// TwinCAT 3 PLC project SPS_3
// ProgramVersion: 3.1.4026.10
// CompilerDefines: VISU_USEPROPERTYINFO
// libraries:
//   Tc2_ModbusRTU, * (Beckhoff Automation GmbH)
//   Tc2_Standard, * (Beckhoff Automation GmbH)
//   Tc2_System, * (Beckhoff Automation GmbH)
//   Tc2_TcpIp, * (Beckhoff Automation GmbH)
//   Tc2_Utilities, * (Beckhoff Automation GmbH)
// project tree:
//   DUTs/01_Listen/01_Zustände/ eObjectAktorState.TcDUT, eObjectSensorState.TcDUT, eSkillState.TcDUT, eSystemState.TcDUT
//   DUTs/01_Listen/02_Commands/ eSystemCommand.TcDUT
//   DUTs/01_Listen/03_Konfigurationen/ eRobMoveType.TcDUT, eRobPosType.TcDUT
//   DUTs/02_Schnittstellen/01_Skills/ I_Skill.TcIO (not stored), I_Skill_RoboterErweitert.TcIO, I_Skill_SmartGreifer.TcIO, I_Skill_Roboter.TcIO
//   DUTs/02_Schnittstellen/02_Objekte/ I_Objekt_Kraftsensor.TcIO (not stored), I_Objekt_Roboter.TcIO, I_Objekt_SmartGreifer.TcIO
//   DUTs/02_Schnittstellen/03_Sequenz/ I_Sequenz.TcIO
//   DUTs/03_Strukturen/01_Prozessparameter/ sKraftVariablen.TcDUT, sRoboterProzessVariablen.TcDUT, sSmartGreiferProzessVariablen.TcDUT
//   DUTs/03_Strukturen/02_Objektintern/01_FB_Roboter/ sPositionArrays.TcDUT, sPositionValues.TcDUT, sRealTimeData.TcDUT
//   DUTs/03_Strukturen/02_Objektintern/02_FB_Kraftsensor/ Kraftvariablen.TcDUT, Request.TcDUT, Response_Parameters.TcDUT, Response_Values.TcDUT
//   DUTs/03_Strukturen/ SkillInfo.TcDUT
//   DUTs/04_Union/ Array2_Int.TcDUT, Array8_LReal.TcDUT, Int_2Byte.TcDUT, String_Array256.TcDUT
//   / GlobalTextList.TcGTLO, PlcTask.TcTTO, Visualization Manager.TcVMO (not stored), VISU_TASK.TcTTO
//   GVLs/ GVL.TcGVL
//   POUs/00_Funktionsbausteine/ FB_PulseTrigger.TcPOU
//   POUs/01_Prozessmodell/01_Skills/01_V1/00_Basis/ FB_Basis_Skill.TcPOU, FB_SkillReferenz.TcPOU
//   POUs/01_Prozessmodell/01_Skills/01_V1/01_Roboter/ Skill_Position_anfahren.TcPOU, Skill_Position_anfahren_erweitert.TcPOU (not stored)
//   POUs/01_Prozessmodell/01_Skills/01_V1/02_Greifer/ Skill_Greifer_Pos_Anfahren.TcPOU (not stored)
//   POUs/01_Prozessmodell/01_Skills/02_V2/01_Roboter/ FB_SkillBasis.TcPOU, Skill_R_P2P.TcPOU
//   POUs/01_Prozessmodell/02_Sequenzen/00_Basis/ FB_Basis.TcPOU
//   POUs/01_Prozessmodell/02_Sequenzen/01_Version_1/ Seq_Ausrichten.TcPOU, Seq_Ausrichten_MPlate.TcPOU, Seq_Ausrichten_Plates.TcPOU, Seq_Get_Part.TcPOU, Seq_Set_MPlate.TcPOU, Seq_Set_Plate_1.TcPOU (not stored), Seq_Set_Plate_2.TcPOU (not stored)
//   POUs/01_Prozessmodell/02_Sequenzen/02_Version_2/ Seq_Teile_Hohlen.TcPOU
//   POUs/01_Prozessmodell/03_Arbeitsplan/ AP_V1.TcPOU, AP_V2.TcPOU, AP_V2_1.TcPOU
//   POUs/01_Prozessmodell/ SkillSet.TcPOU
//   POUs/02_Anlagenmodell/01_Objektklassen/00_Referenz/ Basis_Objekt.TcPOU, FB_Basis_Objekt_Aktor.TcPOU, FB_Basis_Objekt_Sensor.TcPOU
//   POUs/02_Anlagenmodell/01_Objektklassen/ FB_Kraftsensor_V2.TcPOU, FB_Roboter.TcPOU, FB_SmartGreifer.TcPOU
//   POUs/02_Anlagenmodell/ Anlage.TcPOU
//   POUs/03_Systemmodell/ Systemparameter.TcPOU, Zustandshandling.TcPOU
//   POUs/ MAIN.TcPOU, PunkteZuweisung_Temp.TcPOU
//   VISUs/ Visualization.TcVIS
// real-time tasks:
//   TASK VISU_TASK: cycle T#200000us, priority 30, ADS port 351
//   TASK PlcTask2: cycle T#10ms, priority 22, ADS port 353
// I/O:
//   DEVICE Gerät 1 (EtherCAT), AmsNetId 147.87.172.51.2.1
//     Box 1 (BK1120)
// variable links:
//   SPS_3/SPS_3 Instance <-> Device 1 (EtherCAT)/Box 1 (BK1120)
//     PlcTask Inputs/Anlage.Gripper.Communication.InData/D[{0..21}] <-> Term 2 (KL6041)/Channel 1/Data In {0..21}  (22 links)
//     PlcTask Inputs/Anlage.Gripper.Communication.InData/Status <-> Term 2 (KL6041)/Channel 1/Status
//     PlcTask Outputs/Anlage.Gripper.Communication.OutData/Ctrl <-> Term 2 (KL6041)/Channel 1/Ctrl
//     PlcTask Outputs/Anlage.Gripper.Communication.OutData/D[{0..21}] <-> Term 2 (KL6041)/Channel 1/Data Out {0..21}  (22 links)

CONFIGURATION SPS_3
    RESOURCE PLC ON TwinCAT3
        TASK PlcTask(INTERVAL := T#10ms, PRIORITY := 22);
        TASK VISU_TASK(INTERVAL := T#200000us, PRIORITY := 30);
        PROGRAM MAIN WITH PlcTask : MAIN;
        PROGRAM VisuElems_Visu_Prg WITH VISU_TASK : VisuElems.Visu_Prg;
    END_RESOURCE
END_CONFIGURATION

// ---- DUTs/01_Listen/01_Zustände/eObjectAktorState.TcDUT
{attribute 'qualified_only'}
{attribute 'strict'}
{attribute 'to_string'}
TYPE eObjectAktorState :
(
	AUS 					:= 0,				// Das Objekt ist ausgeschalten
	BEREIT 					:= 1,				// Das Objekt ist eingeschalten und bereit
	MANUELL					:= 2,				// Das Objekt befindet sich im Manuell-Modus
	LAUFEND 				:= 3,				// Das Objekt ist aktiv
	ABGESCHLOSSEN_INTERN 	:= 4,				// Das Objekt hat den Prozess durchgeführt und hat selbständig gestoppt
	ABGESCHLOSSEN_EXTERN	:= 5,				// Das Objekt wurde durch den Skill gestoppt (ERREICHT / LIMIT)
	GESTOPPT 				:= 6,				// Das Objekt wurde durch das System gestoppt
	FEHLER					:= 7				// Es gibt einen Fehler bezüglich des Objektes
);
END_TYPE

// ---- DUTs/01_Listen/01_Zustände/eObjectSensorState.TcDUT
{attribute 'qualified_only'}
{attribute 'strict'}
{attribute 'to_string'}
TYPE eObjectSensorState :
(
	AUS 					:= 0,				// Das Objekt ist ausgeschalten
	LAUFEND 				:= 1,				// Das Objekt ist aktiv
	FEHLER					:= 2				// Es gibt einen Fehler bezüglich des Objektes
);
END_TYPE

// ---- DUTs/01_Listen/01_Zustände/eSkillState.TcDUT
{attribute 'qualified_only'}
{attribute 'strict'}
{attribute 'to_string'}
TYPE eSkillState :
(
	BEREIT	 		:= 0,				// Der Skill ist bereit einen Prozess auszuführen (Startzustand)
	LAUFEND 		:= 1,				// Der Skill führt einen Prozess aus
	ABGESCHLOSSEN 	:= 2,				// Der Prozess wurde abgeschlossen (Durch Objekt abgeschlossen)
	FEHLER			:= 3,				// Es gibt einen Fehler bezüglich des Prozesses 
	LIMITE			:= 4,				// Grenzwert wurde überschritten und Prozess wurde abgebrochen
	ERREICHT		:= 5				// Prozessziel wurde erreicht und Prozess wurde durch Skill beendet  
);	
END_TYPE

// ---- DUTs/01_Listen/01_Zustände/eSystemState.TcDUT
{attribute 'qualified_only'}
{attribute 'strict'}
{attribute 'to_string'}
TYPE eSystemState :
(
	AUS 			:= 0,				// Das System ist ausgeschalten
	BEREIT 			:= 1,				// Das System ist eingeschalten und bereit einen Prozess durchzuführen
	LAUFEND 		:= 2,				// Ein Prozess wird ausgeführt
	GESTOPPT		:= 3,				// Ein Prozess wurde gestoppt
	FEHLER			:= 4				// Es gibt einen Fehler im System 
);
END_TYPE

// ---- DUTs/01_Listen/02_Commands/eSystemCommand.TcDUT
{attribute 'qualified_only'}
{attribute 'strict'}
{attribute 'to_string'}
TYPE eSystemCommand :
(
	KEINE		:= 0,
	AUSCHALTEN 	:= 1,
	EINSCHALTEN := 2,
	STOPPEN		:= 3,
	RESETTEN	:= 4
);
END_TYPE

// ---- DUTs/01_Listen/03_Konfigurationen/eRobMoveType.TcDUT
{attribute 'qualified_only'}
{attribute 'strict'}
{attribute 'to_string'}
TYPE eRobMoveType :
(
	LinearToolSpace 			:= 0,		// Move to position (linear in tool-space)
	LinearJointSpace 			:= 1,		// Move to position (linear in joint-space)
	CircularToolSpace 			:= 2,		// Move Circular: Move to position (circular in tool-space)
	BlendCircularMoveLinear		:= 3		// Move Process
);
END_TYPE

// ---- DUTs/01_Listen/03_Konfigurationen/eRobPosType.TcDUT
{attribute 'qualified_only'}
{attribute 'strict'}
{attribute 'to_string'}
TYPE eRobPosType :
(
	Absolut := 0,			// Absolute Bewegung bezogen auf Basis-Koordinatensystem
	Relativ := 1			// Relative Bewegung bezogen auf aktuelle Position
);
END_TYPE

// ---- DUTs/03_Strukturen/01_Prozessparameter/sKraftVariablen.TcDUT
TYPE sKraftVariablen :
STRUCT
	Fx					:LREAL;							// Kraft in X-Richtung 
	Fy					:LREAL;							// Kraft in Y-Richtung 
	Fz					:LREAL;							// Kraft in Z-Richtung 
END_STRUCT
END_TYPE

// ---- DUTs/03_Strukturen/01_Prozessparameter/sRoboterProzessVariablen.TcDUT

TYPE sRoboterProzessVariablen :
STRUCT
	q1					:LREAL;				// X-Koordinate oder Gelenkwinkel 1
	q2					:LREAL;				// Y-Koordinate oder Gelenkwinkel 2
	q3					:LREAL;				// Z-Koordinate oder Gelenkwinkel 3
	q4					:LREAL;				// Orintierung um X-Achse oder Gelenkwinkel 4
	q5					:LREAL;				// Orientierung um Y-Achse oder Gelenkwinkel 5
	q6					:LREAL;				// Orientierung um Z-Achse oder Gelenkwinkel 6
	v					:LREAL;				// Geschwindigkeit
	a					:LREAL;				// Beschleunigung
	PosTyp				:eRobPosType;		// Position-Typ definieren (Absolut / Relativ)		
	MoveTyp				:eRobMoveType;		// Bewegungsart definieren (Linear / Circular etc.)
END_STRUCT
END_TYPE

// ---- DUTs/03_Strukturen/01_Prozessparameter/sSmartGreiferProzessVariablen.TcDUT
TYPE sSmartGreiferProzessVariablen :
STRUCT
	Pos				:USINT;			// Position von Greifer in mm
	Geschw			:USINT;			// Geschwindigkeit in %
	F				:USINT;			// Kraft in %
END_STRUCT
	
END_TYPE

// ---- DUTs/03_Strukturen/02_Objektintern/01_FB_Roboter/sPositionArrays.TcDUT
TYPE sPositionArrays :
STRUCT
	q1		: ARRAY[0..7] OF BYTE;
	q2		: ARRAY[0..7] OF BYTE;
	q3		: ARRAY[0..7] OF BYTE;
	q4		: ARRAY[0..7] OF BYTE;
	q5		: ARRAY[0..7] OF BYTE;
	q6		: ARRAY[0..7] OF BYTE;
END_STRUCT
END_TYPE

// ---- DUTs/03_Strukturen/02_Objektintern/01_FB_Roboter/sPositionValues.TcDUT
TYPE sPositionValues :
STRUCT
	q1			:LREAL;
	q2			:LREAL;
	q3			:LREAL;
	q4			:LREAL;
	q5			:LREAL;
	q6			:LREAL;
END_STRUCT
END_TYPE

// ---- DUTs/03_Strukturen/02_Objektintern/01_FB_Roboter/sRealTimeData.TcDUT
TYPE sRealTimeData :
STRUCT
	messageSize 				: ARRAY[0..3] OF BYTE;
	
	timestamp 					: ARRAY[0..7] OF BYTE;
	
	//qTarget 					: ARRAY[0..47] OF BYTE;
	qTargetQ1 					: ARRAY[0..7] OF BYTE;
	qTargetQ2 					: ARRAY[0..7] OF BYTE;
	qTargetQ3 					: ARRAY[0..7] OF BYTE;
	qTargetQ4 					: ARRAY[0..7] OF BYTE;
	qTargetQ5 					: ARRAY[0..7] OF BYTE;
	qTargetQ6 					: ARRAY[0..7] OF BYTE;
	
	qdTarget 					: ARRAY[0..47] OF BYTE;
	
	qddTarget 					: ARRAY[0..47] OF BYTE;
	
	iTarget 					: ARRAY[0..47] OF BYTE;
	
	mTarget 					: ARRAY[0..47] OF BYTE;
	
	//qActual 					: ARRAY[0..47] OF BYTE;
	qActualQ1 					: ARRAY[0..7] OF BYTE;
	qActualQ2 					: ARRAY[0..7] OF BYTE;
	qActualQ3 					: ARRAY[0..7] OF BYTE;
	qActualQ4 					: ARRAY[0..7] OF BYTE;
	qActualQ5 					: ARRAY[0..7] OF BYTE;
	qActualQ6 					: ARRAY[0..7] OF BYTE;
	
	//qdActual 					: ARRAY[0..47] OF BYTE;
	qdActualQ1 					: ARRAY[0..7] OF BYTE;
	qdActualQ2 					: ARRAY[0..7] OF BYTE;
	qdActualQ3 					: ARRAY[0..7] OF BYTE;
	qdActualQ4 					: ARRAY[0..7] OF BYTE;
	qdActualQ5 					: ARRAY[0..7] OF BYTE;
	qdActualQ6 					: ARRAY[0..7] OF BYTE;
	
	iActual 					: ARRAY[0..47] OF BYTE;
	
	toolAccelerometerValues 	: ARRAY[0..23] OF BYTE;
	
	unused_1					: ARRAY[0..119] OF BYTE;
	
	tcpForce 					: ARRAY[0..47] OF BYTE;
	
	//toolVector 					: ARRAY[0..47] OF BYTE;
	toolVectorQ1 				: ARRAY[0..7] OF BYTE;
	toolVectorQ2 				: ARRAY[0..7] OF BYTE;
	toolVectorQ3 				: ARRAY[0..7] OF BYTE;
	toolVectorQ4 				: ARRAY[0..7] OF BYTE;
	toolVectorQ5 				: ARRAY[0..7] OF BYTE;
	toolVectorQ6 				: ARRAY[0..7] OF BYTE;
	
	tcpSpeed 					: ARRAY[0..47] OF BYTE;
	
	digitalInputBits 			: ARRAY[0..7] OF BYTE;
	
	unused_2					: ARRAY[0..119] OF BYTE;
END_STRUCT
END_TYPE

// ---- DUTs/03_Strukturen/02_Objektintern/02_FB_Kraftsensor/Kraftvariablen.TcDUT

TYPE Kraftvariablen :
STRUCT
	Fx					:LREAL;							// Kraft in X-Richtung 
	Fy					:LREAL;							// Kraft in Y-Richtung 
	Fz					:LREAL;							// Kraft in Z-Richtung 
	Tx					:LREAL;							// Moment auf X-Achse 
	Ty					:LREAL;							// Moment auf Y-Achse 
	Tz					:LREAL;							// Moment auf Z-Achse 
END_STRUCT
END_TYPE

// ---- DUTs/03_Strukturen/02_Objektintern/02_FB_Kraftsensor/Request.TcDUT
TYPE Request :
STRUCT
	Command			:UINT;		// Value according to the command table
	Data			:ARRAY[0..18] OF UINT := [0];		
END_STRUCT
END_TYPE

// ---- DUTs/03_Strukturen/02_Objektintern/02_FB_Kraftsensor/Response_Parameters.TcDUT
TYPE Response_Parameters :
STRUCT
	Header				:UINT;			// Fixed 0x1234
	Unit_Force			:USINT;			// The unit of the calculated Force values
	Unit_Torque			:USINT;			// The unit of the calculated Torque values
	CPF					:UDINT;			// Counts per Force value
	CPT					:UDINT;			// Counts per Torque value
	ScaleFactorFx		:UINT;			// Additional scaling factor (for the Fx,Fy,Fz,Tx,Ty,Tz)
	ScaleFactorFy		:UINT;			// Additional scaling factor (for the Fx,Fy,Fz,Tx,Ty,Tz)
	ScaleFactorFz		:UINT;			// Additional scaling factor (for the Fx,Fy,Fz,Tx,Ty,Tz)
	ScaleFactorTx		:UINT;			// Additional scaling factor (for the Fx,Fy,Fz,Tx,Ty,Tz)
	ScaleFactorTy		:UINT;			// Additional scaling factor (for the Fx,Fy,Fz,Tx,Ty,Tz)
	ScaleFactorTz		:UINT;			// Additional scaling factor (for the Fx,Fy,Fz,Tx,Ty,Tz)
END_STRUCT
END_TYPE

// ---- DUTs/03_Strukturen/02_Objektintern/02_FB_Kraftsensor/Response_Values.TcDUT
TYPE Response_Values :
STRUCT
	Header				:UINT;			// Fixed 0x1234
	Status				:UINT;			// Status word of the sensor and Compute Box
	Fx					:INT;			// X-axis force in 32 bit Counts*
	Fy					:INT;			// Y-axis force in 32 bit Counts*
	Fz					:INT;			// Z-axis force in 32 bit Counts*
	Tx					:INT;			// X-axis torque in 32 bit Counts* (0 if not available)
	Ty					:INT;			// Y-axis torque in 32 bit Counts* (0 if not available)
	Tz					:INT;			// Z-axis torque in 32 bit Counts* (0 if not available)
END_STRUCT
END_TYPE

// ---- DUTs/03_Strukturen/SkillInfo.TcDUT
TYPE SkillInfo :
STRUCT
	iState			:eSkillState;
	Data			:sRoboterProzessVariablen;
	iStateObj		:eObjectAktorState;
	DataObj			:sRoboterProzessVariablen;
END_STRUCT
END_TYPE

// ---- DUTs/04_Union/Array2_Int.TcDUT
TYPE Array2_Int :
UNION
	arrByte 		:ARRAY[0..1] OF BYTE;
	sValue			:INT; 
END_UNION
END_TYPE

// ---- DUTs/04_Union/Array8_LReal.TcDUT
TYPE Array8_LReal :
UNION
	arrByte			:ARRAY[0..7] OF BYTE;
	rValue			:LREAL;
END_UNION
END_TYPE

// ---- DUTs/04_Union/Int_2Byte.TcDUT
TYPE Int_2Byte :
UNION
	sValue			:INT; 
	arrByte 		:ARRAY[0..1] OF BYTE;
END_UNION
END_TYPE

// ---- DUTs/04_Union/String_Array256.TcDUT
TYPE String_Array256 :
UNION
	sValue			:STRING; 
	arrByte 		:ARRAY[0..255] OF BYTE;
END_UNION
END_TYPE

// ---- GVLs/GVL.TcGVL
{attribute 'qualified_only'}
VAR_GLOBAL
	// Schnittstellenvariablen 
		// System: 
		SystemState								:eSystemState; 
		SystemCommand							:eSystemCommand; 
		ErrorID									:INT;
		
		// Kontrollvariablen: 
		Reset									:BOOL;
		Execute									:BOOL;
		
		// Prozessvariablen
		eKraftLimitValue						:sKraftVariablen;
		eKraftErreichtValue						:sKraftVariablen;
		
		
		// SkillStates
		
		// ObjectStates
		Robot_State								:eObjectAktorState;
		Greifer_State							:eObjectAktorState;
		Sensor_State							:eObjectSensorState;
		
		// Testvariablen
		CountSkillStart							:INT;
		CountSkill								:INT;
		CountObjectStart						:INT;
		CountObject								:INT;
		TestCount								:INT;
		MethodeState							:INT;
		SkillArray								:ARRAY[0..10] OF sRoboterProzessVariablen;
		ObjectArray								:ARRAY[0..10] OF STRING;
		skillInfo 								:ARRAY[0..50] OF SkillInfo;
		InfoCountSkill							:INT;
		PulseNrArray							:Array[0..10] OF INT;
END_VAR

// ---- DUTs/02_Schnittstellen/01_Skills/I_Skill_RoboterErweitert.TcIO
INTERFACE I_Skill_RoboterErweitert

METHOD M_Reset : BOOL
VAR_INPUT
END_VAR
END_METHOD

METHOD M_Start : BOOL
VAR_INPUT
END_VAR
END_METHOD

METHOD M_Stop : BOOL
VAR_INPUT
END_VAR
END_METHOD

PROPERTY P_Erreicht : sKraftVariablen
SET
END_SET
END_PROPERTY

PROPERTY P_Limit : sKraftVariablen
SET
END_SET
END_PROPERTY

PROPERTY P_RobotParam : sRoboterProzessVariablen
SET
END_SET
END_PROPERTY

PROPERTY P_State : eSkillState
GET
END_GET
END_PROPERTY

END_INTERFACE

// ---- DUTs/02_Schnittstellen/01_Skills/I_Skill_SmartGreifer.TcIO
INTERFACE I_Skill_SmartGreifer

METHOD M_Reset : BOOL
VAR_INPUT
END_VAR
END_METHOD

METHOD M_Start : BOOL
VAR_INPUT
END_VAR
END_METHOD

METHOD M_Stop : BOOL
VAR_INPUT
END_VAR
END_METHOD

PROPERTY P_SGripperParam : sSmartGreiferProzessVariablen
SET
END_SET
END_PROPERTY

PROPERTY P_State : eSkillState
GET
END_GET
END_PROPERTY

END_INTERFACE

// ---- DUTs/02_Schnittstellen/01_Skills/I_Skill_Roboter.TcIO
INTERFACE I_Skill_Roboter

METHOD M_Reset : BOOL
VAR_INPUT
END_VAR
END_METHOD

METHOD M_Start : BOOL
VAR_INPUT
END_VAR
END_METHOD

METHOD M_Stop : BOOL
VAR_INPUT
END_VAR
END_METHOD

PROPERTY P_RobotParam : sRoboterProzessVariablen
SET
END_SET
END_PROPERTY

PROPERTY P_State : eSkillState
GET
END_GET
END_PROPERTY

END_INTERFACE

// ---- DUTs/02_Schnittstellen/02_Objekte/I_Objekt_Roboter.TcIO
INTERFACE I_Objekt_Roboter

METHOD M_Reset : BOOL
VAR_INPUT
END_VAR
END_METHOD

METHOD M_Start : BOOL
VAR_INPUT
END_VAR
END_METHOD

METHOD M_Stop : BOOL
VAR_INPUT
END_VAR
END_METHOD

PROPERTY P_Prozessparameter : sRoboterProzessVariablen
SET
END_SET
END_PROPERTY

PROPERTY P_State : eObjectAktorState
GET
END_GET
END_PROPERTY

PROPERTY Test_Param : sRoboterProzessVariablen
GET
END_GET
END_PROPERTY

END_INTERFACE

// ---- DUTs/02_Schnittstellen/02_Objekte/I_Objekt_SmartGreifer.TcIO
INTERFACE I_Objekt_SmartGreifer

METHOD M_Reset : BOOL
VAR_INPUT
END_VAR
END_METHOD

METHOD M_Start : BOOL
VAR_INPUT
END_VAR
END_METHOD

METHOD M_Stop : BOOL
VAR_INPUT
END_VAR
END_METHOD

PROPERTY P_Prozessparameter : sSmartGreiferProzessVariablen
SET
END_SET
END_PROPERTY

PROPERTY P_State : eObjectAktorState
GET
END_GET
END_PROPERTY

END_INTERFACE

// ---- DUTs/02_Schnittstellen/03_Sequenz/I_Sequenz.TcIO
INTERFACE I_Sequenz

METHOD M_Reset : BOOL
VAR_INPUT
END_VAR
END_METHOD

METHOD M_Start : BOOL
VAR_INPUT
END_VAR
END_METHOD

METHOD M_Stop : BOOL
VAR_INPUT
END_VAR
END_METHOD

PROPERTY P_Finished : BOOL
GET
END_GET
END_PROPERTY

PROPERTY P_State : INT
GET
END_GET
END_PROPERTY

END_INTERFACE

// ---- POUs/MAIN.TcPOU
PROGRAM MAIN
VAR
END_VAR

// Aufrufen der Objekte
Anlage();
// Aufrufen der Skills (Im Moment nur für V1 verwendet)
//SkillSet();
// Aufrufen der Systenparameterzuweisung 
Systemparameter();
// Aufrunfen des Zustandshandlings
Zustandshandling();
// Temporäre Punktedatenbank
PunkteZuweisung_Temp();

// Aufrufen von Testablauf
AP_V2();

END_PROGRAM

// ---- POUs/02_Anlagenmodell/Anlage.TcPOU
PROGRAM Anlage
VAR_INPUT
	UR5				:FB_Roboter;
	Gripper			:FB_SmartGreifer;
	HEX_E_V2		:FB_Kraftsensor_V2;
END_VAR

VAR
END_VAR

UR5(
    eSysState := GVL.SystemState,
    eSysCommand := GVL.SystemCommand,
    sIP := '192.168.1.100',
    iPort_Prim := 30002,
    iPort_RT := 30003); // FB_Roboter
Gripper(eSysState := GVL.SystemState, eSysCommand := GVL.SystemCommand); // FB_SmartGreifer
HEX_E_V2(
    eSysState := GVL.SystemState,
    eSysCommand := GVL.SystemCommand,
    sIP := '192.168.1.10',
    iPort := 49151); // FB_Kraftsensor_V2

END_PROGRAM

// ---- POUs/02_Anlagenmodell/01_Objektklassen/FB_Roboter.TcPOU
FUNCTION_BLOCK FB_Roboter EXTENDS FB_Basis_Objekt_Aktor IMPLEMENTS I_Objekt_Roboter
VAR_INPUT
	// Kommunikationsvariablen
	sIP						:T_IPv4Addr;
	iPort_Prim				:UINT;
	iPort_RT				:UINT;
END_VAR

VAR_OUTPUT
END_VAR

VAR
	// Instanziierung von Kommunikationsbausteine
	Connect					:FB_SocketConnect;
	Disconnect				:FB_SocketCloseALL;
	Send_START				:FB_SocketSend;
	Send_STOP				:FB_SocketSend;
	Connect_RT				:FB_SocketConnect;
	Receive_RT				:FB_SocketReceive;
	Disconnect_RT			:FB_SocketClose;
	
	// Kommunikationsvariablen
	sSrvNetId   			:T_AmsNetId := '';
	tTimeout    			:TIME := T#45S;(*!!!*)
	hSocket    				:T_HSOCKET;
	hSocket_RT    			:T_HSOCKET;
	
	// Managementvariablen
	bEingeschalten 			:BOOL;
	bAusgeschalten			:BOOL;
	bAmStarten				:BOOL;
	bGestartet				:BOOL;
	bAmStoppen				:BOOL;
	bGestoppt				:BOOL;
	
	bStopCommand			:BOOL;
	bTurnedOn 				:BOOL;
	
	bBewegungStoppen		:BOOL;
	
	Delay_1					:TON;
	Execute_TON1			:BOOL;
	Delay_2					:TON;
	
	bQ1						:BOOL;
	bQ2						:BOOL;
	bQ3						:BOOL;
	bQ4						:BOOL;
	bQ5						:BOOL;
	bQ6						:BOOL;
	
	bVQ1					:BOOL;
	bVQ2					:BOOL;
	bVQ3					:BOOL;
	bVQ4					:BOOL;
	bVQ5					:BOOL;
	bVQ6					:BOOL;
	
	// RealTimeDatenerfassung
	RT_State				:INT;							// RealTime-State-Variable
	ReceivedData			:sRealTimedata;					// Erhaltene Daten von Roboter
	nRecBytes				:UDINT;							// Anzahl der erhaltenen Bytes
	
	JointPositions			:sPositionValues;				// Ausgelesene aktuelle Joint-Positonen-Byte
	JointSpeed				:sPositionValues;				// Ausgelesene aktuelle Joint-Geschwindigkeit-Byte
	ToolPosition			:sPositionValues;				// Ausgelesene aktuelle Tool-Positonen-Byte
	
	TempJointPosRev			:sPositionArrays;				// Ausgelesene aktuelle Joint-Positonen-Byte (Reversed)
	TempJointVRev			:sPositionArrays;				// Ausgelesene aktuelle Joint-Geschwindigkeit-Byte (Reversed)	
	TempToolPosRev			:sPositionArrays;				// Ausgelesene aktuelle Tool-Positonen-Byte(Reversed)
	
	Joint					:Array8_LReal;					// Aktuelle Joint-Positonen
	JSpeed					:Array8_LReal;					// Aktuelle Joint-Geschwindgeit
	Tool					:Array8_LReal;					// Aktuelle Tool-Positionen
	m						:INT;							// Loop-Variable
	
	// Prozessdaten
	TargetPosition			:sPositionValues;				// Targetpositions
	bSetValues				:BOOL;							// Definiert ob Targetposition noch ermittelt werden muss
	Prozessvariablen		:sRoboterProzessVariablen;
	
	Stateset				:BOOL;
END_VAR

// Instanziierungen
	Connect_RT(sSrvNetId := sSrvNetId,
							sRemoteHost := sIP,
							nRemotePort := iPort_RT,
							tTimeout := tTimeout,
							bError => bFehler,
							nErrId => iErrorID,
							hSocket => hSocket_RT);	
							
	Send_START(sSrvNetId := sSrvNetId,
			hSocket := hSocket,
			tTimeout := tTimeout,
			bError => bFehler,
			nErrId => iErrorID);
	Send_STOP(sSrvNetId := sSrvNetId,
			hSocket := hSocket,
			tTimeout := tTimeout,
			bError => bFehler,
			nErrId => iErrorID);
							
	Receive_RT(sSrvNetId := sSrvNetId,
							hSocket := hSocket_RT,
							cbLen := SIZEOF(ReceivedData),
							pDest := ADR(ReceivedData),
							tTimeout := tTimeout,
							bError => bFehler,
							nErrId => iErrorID,
							nRecBytes => nRecBytes);
							
	Disconnect_RT(sSrvNetId := sSrvNetId,
							hSocket := hSocket_RT,
							tTimeout := tTimeout,
							bError => bFehler,
							nErrId => iErrorID);
	
	Delay_1(IN := Execute_TON1, PT := T#3MS);
//____________________________________________________________________________________________
// Input-Command-Verwaltung
	// System
	IF eSysCommand = 2 AND iState = 0 THEN			// Objekt einschalten
		bEinschalten := TRUE;
	ELSE 
		bEinschalten := FALSE;
	END_IF
	
	IF eSysCommand = 1 AND iState = 1 THEN			// Objekt ausschalten
		bAusschalten := TRUE;		
	ELSE 
		bAusschalten := FALSE;		
	END_IF
	
	IF eSysCommand = 3 THEN							// Objekt beendet Prozess
		bStoppen := TRUE;
	ELSE
		bStoppen := FALSE;
	END_IF
	
	IF eSysCommand = 4 THEN							// System resettet Objekt
		bResettenSystem := TRUE;
	ELSE
		bResettenSystem := FALSE;
	END_IF
	
	
//____________________________________________________________________________________________
// Interner Methodenaufruf (Durch System oder Skill)
IF bEinschalten THEN
	bEingeschalten := M_Verbinden();
	bTurnedOn := TRUE;
ELSE 
	bEingeschalten := FALSE;
END_IF

IF bAusschalten THEN
	bAusgeschalten := M_Trennen();
	bTurnedOn := FALSE;
	RT_State := 0;
ELSE 
	bAusgeschalten := FALSE;
END_IF

//____________________________________________________________________________________________
// Datenerfassungsprozess
IF bTurnedOn THEN
	CASE RT_State OF 
		0:	// Connect to RealTimePort
				Connect_RT(bExecute := TRUE);			
					
				IF NOT Connect_RT.bBusy AND NOT Connect_RT.bError THEN
					Connect_RT.bExecute := FALSE;
					RT_State := 1;
				END_IF
		
		1:	// Get Data 
				Receive_RT(bExecute := TRUE);
			
				IF NOT Receive_RT.bBusy AND NOT Receive_RT.bError THEN
					Receive_RT.bExecute := FALSE;
					RT_State := 2;
				END_IF
				
		2:	// Use Data
				m := 0;
		
				// Reverse Array
				FOR m := 0 TO 7 DO
					TempJointPosRev.q1[m] := ReceivedData.qActualQ1[7 - m];
					TempJointPosRev.q2[m] := ReceivedData.qActualQ2[7 - m];
					TempJointPosRev.q3[m] := ReceivedData.qActualQ3[7 - m];
					TempJointPosRev.q4[m] := ReceivedData.qActualQ4[7 - m];
					TempJointPosRev.q5[m] := ReceivedData.qActualQ5[7 - m];
					TempJointPosRev.q6[m] := ReceivedData.qActualQ6[7 - m];
					
					TempJointVRev.q1[m] := ReceivedData.qdActualQ1[7 - m];
					TempJointVRev.q2[m] := ReceivedData.qdActualQ2[7 - m];
					TempJointVRev.q3[m] := ReceivedData.qdActualQ3[7 - m];
					TempJointVRev.q4[m] := ReceivedData.qdActualQ4[7 - m];
					TempJointVRev.q5[m] := ReceivedData.qdActualQ5[7 - m];
					TempJointVRev.q6[m] := ReceivedData.qdActualQ6[7 - m];
					
					TempToolPosRev.q1[m] := ReceivedData.toolVectorQ1[7 - m];
					TempToolPosRev.q2[m] := ReceivedData.toolVectorQ2[7 - m];
					TempToolPosRev.q3[m] := ReceivedData.toolVectorQ3[7 - m];
					TempToolPosRev.q4[m] := ReceivedData.toolVectorQ4[7 - m];
					TempToolPosRev.q5[m] := ReceivedData.toolVectorQ5[7 - m];
					TempToolPosRev.q6[m] := ReceivedData.toolVectorQ6[7 - m];
				END_FOR
			
				Joint.arrByte := TempJointPosRev.q1;
				JointPositions.q1 := RAD_TO_DEG(Joint.rValue);
				Joint.arrByte := TempJointPosRev.q2;
				JointPositions.q2 := RAD_TO_DEG(Joint.rValue);
				Joint.arrByte := TempJointPosRev.q3;
				JointPositions.q3 := RAD_TO_DEG(Joint.rValue);
				Joint.arrByte := TempJointPosRev.q4;
				JointPositions.q4 := RAD_TO_DEG(Joint.rValue);
				Joint.arrByte := TempJointPosRev.q5;
				JointPositions.q5 := RAD_TO_DEG(Joint.rValue);
				Joint.arrByte := TempJointPosRev.q6;
				JointPositions.q6 := RAD_TO_DEG(Joint.rValue);
				
				JSpeed.arrByte := TempJointVRev.q1;
				JointSpeed.q1 := JSpeed.rValue;
				JSpeed.arrByte := TempJointVRev.q2;
				JointSpeed.q2 := JSpeed.rValue;
				JSpeed.arrByte := TempJointVRev.q3;
				JointSpeed.q3 := JSpeed.rValue;
				JSpeed.arrByte := TempJointVRev.q4;
				JointSpeed.q4 := JSpeed.rValue;
				JSpeed.arrByte := TempJointVRev.q5;
				JointSpeed.q5 := JSpeed.rValue;
				JSpeed.arrByte := TempJointVRev.q6;
				JointSpeed.q6 := JSpeed.rValue;
				
				Tool.arrByte := TempToolPosRev.q1;
				ToolPosition.q1 := Tool.rValue;
				Tool.arrByte := TempToolPosRev.q2;
				ToolPosition.q2 := Tool.rValue;
				Tool.arrByte := TempToolPosRev.q3;
				ToolPosition.q3 := Tool.rValue;
				Tool.arrByte := TempToolPosRev.q4;
				ToolPosition.q4 := RAD_TO_DEG(Tool.rValue);
				Tool.arrByte := TempToolPosRev.q5;
				ToolPosition.q5 := RAD_TO_DEG(Tool.rValue);
				Tool.arrByte := TempToolPosRev.q6;
				ToolPosition.q6 := RAD_TO_DEG(Tool.rValue);
				
				Delay_2(IN := TRUE, PT := T#0.5S);
				IF Delay_2.Q THEN
					Delay_2(IN := FALSE);
					RT_State := 3;
				END_IF
				
		3:	// Disconnect from RealTimePort
				Disconnect_RT(bExecute := TRUE);
							
				IF NOT Disconnect_RT.bBusy AND NOT Disconnect_RT.bError THEN
					Disconnect_RT.bExecute := FALSE;
					RT_State := 0;
				END_IF
		
	END_CASE
END_IF
//____________________________________________________________________________________________
// Zustandsmanagement

IF bFehler THEN 
	iState := 7;
END_IF

CASE iState OF 
	0: // AUS
		// DO
		
		// TRANSITION
			IF bEingeschalten THEN																	// Verbindung wird aufgebaut
				iState := 1;
			END_IF
			
	//____________________________________________________________________________________________
	1: // BEREIT
		// DO
			IF bStarten THEN
				bAmStarten := M_BewegungZuPosition();
			END_IF
			
			IF bAmStarten  THEN
				bAmStarten := FALSE;	
				bStarten := FALSE;
				Execute_TON1 := TRUE;	 
			END_IF
			
			IF Delay_1.Q THEN
				Execute_TON1 := FALSE;
				bGestartet := TRUE;
			END_IF
		
		// TRANSITION
			IF bAusgeschalten THEN																	// Verbindung wird getrennt
				iState := 0;
			END_IF																									// Manuell-Modus wird eingeschalten
													
			 IF bGestartet THEN																	// Objekt führt Prozessdurch
				bGestartet := FALSE;
				iState := 3;
			 END_IF			
	//____________________________________________________________________________________________
	2: // MANUELL
		// DO
		
		// TRANSITION
	
	//____________________________________________________________________________________________
	3: // LAUFEND
		// DO
			
			// Ermitteln von TargetPosition 
			IF NOT bSetvalues THEN
				// Kartesisch
				IF Prozessvariablen.MoveTyp = 0 OR Prozessvariablen.MoveTyp = 3 THEN
					// Absolut
					IF Prozessvariablen.PosTyp = 0 THEN
						TargetPosition.q1 := Prozessvariablen.q1;
						TargetPosition.q2 := Prozessvariablen.q2;
						TargetPosition.q3 := Prozessvariablen.q3;
						TargetPosition.q4 := Prozessvariablen.q4;
						TargetPosition.q5 := Prozessvariablen.q5;
						TargetPosition.q6 := Prozessvariablen.q6;		
					END_IF
										
					// Relativ
					IF Prozessvariablen.PosTyp = 1 THEN
						TargetPosition.q1 := ToolPosition.q1 + Prozessvariablen.q1;
						TargetPosition.q2 := ToolPosition.q2 + Prozessvariablen.q2;
						TargetPosition.q3 := ToolPosition.q3 + Prozessvariablen.q3;
						TargetPosition.q4 := ToolPosition.q4 + Prozessvariablen.q4;
						TargetPosition.q5 := ToolPosition.q5 + Prozessvariablen.q5;
						TargetPosition.q6 := ToolPosition.q6 + Prozessvariablen.q6;
					END_IF
					
				END_IF
				
				// Gelenkwinkel
				IF Prozessvariablen.MoveTyp = 1 THEN
					TargetPosition.q1 := Prozessvariablen.q1;
					TargetPosition.q2 := Prozessvariablen.q2;
					TargetPosition.q3 := Prozessvariablen.q3;
					TargetPosition.q4 := Prozessvariablen.q4;
					TargetPosition.q5 := Prozessvariablen.q5;
					TargetPosition.q6 := Prozessvariablen.q6;	
				END_IF
			
				bSetvalues := TRUE;
			END_IF

			// Vergleich zwischen IST und SOLL
			// Kartesisch
			IF Prozessvariablen.MoveTyp = 0 OR Prozessvariablen.MoveTyp = 3 THEN
				IF ABS(ABS(TargetPosition.q1) - ABS(ToolPosition.q1)) < 0.001 THEN
					bQ1 := TRUE;
				END_IF
				
				IF ABS(ABS(TargetPosition.q2) - ABS(ToolPosition.q2)) < 0.001 THEN
					bQ2 := TRUE;
				END_IF
				
				IF ABS(ABS(TargetPosition.q3) - ABS(ToolPosition.q3)) < 0.001 THEN
					bQ3 := TRUE;
				END_IF
				
				IF ABS(ABS(TargetPosition.q4) - ABS(ToolPosition.q4)) < 2 THEN
					bQ4 := TRUE;
				END_IF
				
				IF ABS(ABS(TargetPosition.q5) - ABS(ToolPosition.q5)) < 1 THEN
					bQ5 := TRUE;
				END_IF
				
				IF ABS(ABS(TargetPosition.q6) - ABS(ToolPosition.q6)) < 1 THEN
					bQ6 := TRUE;
				END_IF
			END_IF
			
			// Gelenkwinkel
			IF Prozessvariablen.MoveTyp = 1 THEN
				IF ABS(ABS(TargetPosition.q1) - ABS(JointPositions.q1)) < 1 THEN
					bQ1 := TRUE;
				END_IF
				
				IF ABS(ABS(TargetPosition.q2) - ABS(JointPositions.q2)) < 1 THEN
					bQ2 := TRUE;
				END_IF
				
				IF ABS(ABS(TargetPosition.q3) - ABS(JointPositions.q3)) < 1 THEN
					bQ3 := TRUE;
				END_IF
				
				IF ABS(ABS(TargetPosition.q4) - ABS(JointPositions.q4)) < 1 THEN
					bQ4 := TRUE;
				END_IF
				
				IF ABS(ABS(TargetPosition.q5) - ABS(JointPositions.q5)) < 1 THEN
					bQ5 := TRUE;
				END_IF
				
				IF ABS(ABS(TargetPosition.q6) - ABS(JointPositions.q6)) < 1 THEN
					bQ6 := TRUE;
				END_IF
			END_IF
			
			// Objekt schliessen Prozess ab
			IF bQ1 AND bQ2 AND bQ3 AND bQ4 AND bQ5 AND bQ6 THEN										// Abgeschlossener Prozess
				
				bQ1 := FALSE;
				bQ2 := FALSE;
				bQ3 := FALSE;
				bQ4 := FALSE;
				bQ5 := FALSE;
				bQ6 := FALSE;
				bObjektFertig := TRUE;
			END_IF
			
				
			// Objekt wird gestoppt durch Skill
			IF bSkillFertig THEN
				
				bQ1 := FALSE;
				bQ2 := FALSE;
				bQ3 := FALSE;
				bQ4 := FALSE;
				bQ5 := FALSE;
				bQ6 := FALSE;
				bSetvalues := FALSE;
				
				bBewegungStoppen := M_BewegungStoppen();
				
				IF bBewegungStoppen THEN
					bBewegungStoppen := FALSE;
					bAmStoppen := TRUE;
				END_IF
			END_IF 
			
			// Objekt wird gestoppt durch System
			IF bStoppen THEN
				
				bQ1 := FALSE;
				bQ2 := FALSE;
				bQ3 := FALSE;
				bQ4 := FALSE;
				bQ5 := FALSE;
				bQ6 := FALSE;
				bSetvalues := FALSE;
				
				bBewegungStoppen := M_BewegungStoppen();
				
				IF bBewegungStoppen THEN
					bBewegungStoppen := FALSE;
					bAmStoppen := TRUE;
				END_IF
			END_IF 
			
			// Stoppprozess
			IF bAmStoppen THEN
				IF JointSpeed.q1 < 0.001 THEN
					bVQ1 := TRUE;
				END_IF
				
				IF JointSpeed.q2 < 0.001 THEN
					bVQ2 := TRUE;
				END_IF
				
				IF JointSpeed.q3 < 0.001 THEN
					bVQ3 := TRUE;
				END_IF
				
				IF JointSpeed.q4 < 0.001 THEN
					bVQ4 := TRUE;
				END_IF
				
				IF JointSpeed.q5 < 0.001 THEN
					bVQ5 := TRUE;
				END_IF
				
				IF JointSpeed.q6 < 0.001 THEN
					bVQ6 := TRUE;
				END_IF
				
				IF bVQ1 AND bVQ2 AND bVQ3 AND bVQ4 AND bVQ5 AND bVQ6 THEN							// Gestoppter Prozess
					bVQ1 := FALSE;	
					bVQ2 := FALSE;	
					bVQ3 := FALSE;	
					bVQ4 := FALSE;	
					bVQ5 := FALSE;	
					bVQ6 := FALSE;	
					
					bAmStoppen := FALSE;
					bGestoppt := TRUE;
					
				END_IF
				
			END_IF
		
		// TRANSITION
			IF bObjektFertig THEN
				bObjektFertig := FALSE;
				bSetvalues := FALSE;
				iState := 4;
			END_IF
			
			IF bGestoppt THEN	
				bGestoppt := FALSE;
				bStopCommand := FALSE;
				
				IF bSkillFertig THEN
					bSkillFertig := FALSE;
					iState := 5;
				END_IF
					
				IF bStoppen THEN
					iState := 6;
				END_IF
					
			END_IF
	
	//____________________________________________________________________________________________
	4: // ABGESCHLOSSEN_INTERN
		// DO
		
		// TRANSITION
			IF bResettenSkill THEN																	// Objekt resetten	
				iState := 1;
			END_IF
	//____________________________________________________________________________________________
	5: // ABGESCHLOSSEN_EXTERN
		// DO																					
		
		// TRANSITION
			IF bResettenSkill THEN																	// Objekt resetten
				iState := 1;
			END_IF
	
	//____________________________________________________________________________________________
	6: // GESTOPPT
		// DO
		
		// TRANSITION
			IF bResettenSystem THEN																	// Objekt resetten
				iState := 1;
			END_IF
	
	//____________________________________________________________________________________________
	7: // FEHLER
		// DO
			
		// TRANSITION
			IF bResettenSystem THEN																	// Objekt resetten
				bFehler	 := FALSE;
				iState := 1;
			END_IF
END_CASE

METHOD M_BewegungStoppen : BOOL
VAR_INPUT
END_VAR
VAR
	stringFormat   		:FB_FormatString;		// Funktion für Stringerstellung	
	a					:INT := 2;

	Command				:T_MaxString;			// Commandstring
	CommandArray		:String_Array256;		// Byte-Array für Kommunikation mit Roboter
END_VAR
stringFormat(sFormat := 'stopj(%d)',
							arg1 := F_INT(a),
							bError => bFehler,
							nErrId => iErrorID,
							sOut => Command);	
							
// VOrbereiten von Array 
	CommandArray.sValue := Command;
	CommandArray.arrByte[LEN(CommandArray.sValue)] := 10;
	
// Senden von Array
	IF NOT bStopCommand THEN
		Send_STOP(cbLen := LEN(CommandArray.sValue),
			pSrc := ADR(CommandArray.arrByte),
			bExecute := TRUE);
			
		bStopCommand := TRUE;
	END_IF
			
	IF NOT Send_STOP.bBusy THEN
		Send_STOP(bExecute := FALSE);
		M_BewegungStoppen := TRUE;
	END_IF
END_METHOD

METHOD M_BewegungZuPosition : BOOL
VAR 
	
	x					:LREAL;				// X-Koordinate
	y					:LREAL;				// Y-Koordinate
	z					:LREAL;				// Z-Koordinate
	rx					:LREAL;				// Orintierung um X-Achse
	ry					:LREAL;				// Orientierung um Y-Achse
	rz					:LREAL;				// Orientierung um Z-Achse
	
	q1					:LREAL;				// Joint-Position 1
	q2					:LREAL;				// Joint-Position 2
	q3					:LREAL;				// Joint-Position 3
	q4					:LREAL;				// Joint-Position 4
	q5					:LREAL;				// Joint-Position 5
	q6					:LREAL;				// Joint-Position 6

	stringFormat   : FB_FormatString;		// Funktion für Stringerstellung

	pose			:T_MaxString;			// Positionsstring
	Command			:T_MaxString;			// Commandstring
	
	CommandArray	:String_Array256;			// Byte-Array für Kommunikation mit Roboter
	
END_VAR
VAR_INPUT
	
END_VAR
// Einfluss von Positionart
	IF Prozessvariablen.PosTyp = 1 THEN		// Relative Bewegung
		
		x := ToolPosition.q1 + Prozessvariablen.q1;
		y := ToolPosition.q2 + Prozessvariablen.q2;
		z := ToolPosition.q3 + Prozessvariablen.q3;
		rx := DEG_TO_RAD(ToolPosition.q4 + Prozessvariablen.q4);
		ry := DEG_TO_RAD(ToolPosition.q5 + Prozessvariablen.q5);
		rz := DEG_TO_RAD(ToolPosition.q6 + Prozessvariablen.q6);
		
	END_IF
	
	IF Prozessvariablen.PosTyp = 0 THEN		// Absolute Bewegung
		
		x := Prozessvariablen.q1;
		y := Prozessvariablen.q2;
		z := Prozessvariablen.q3;
		rx := DEG_TO_RAD(Prozessvariablen.q4);
		ry := DEG_TO_RAD(Prozessvariablen.q5);
		rz := DEG_TO_RAD(Prozessvariablen.q6);
		
	END_IF
	
	stringFormat(sFormat := 'p[%.3f,%.3f,%.3f,%.3f,%.3f,%.3f]',
			arg1 := F_LREAL(x),
			arg2 := F_LREAL(y),
			arg3 := F_LREAL(z),
			arg4 := F_LREAL(rx),
			arg5 := F_LREAL(ry),
			arg6 := F_LREAL(rz),
			bError => bFehler,
			nErrId => iErrorID,
			sOut => pose);

// Einlfuss von Bewegungsart
	IF Prozessvariablen.MoveTyp = 0 THEN			// Move to position (linear in tool-space)
													// movel(pose, a=1.2, v=0.25, t=0, r=0)
		stringFormat(sFormat := 'movel(%s, a=%.2f, v=%.2f)',
							arg1 := F_STRING(pose),
							arg2 := F_LREAL(Prozessvariablen.a),
							arg3 := F_LREAL(Prozessvariablen.v),
							bError => bFehler,
							nErrId => iErrorID,
							sOut => Command);											
	END_IF
	
	IF Prozessvariablen.MoveTyp = 1 THEN			// Move to position (linear in joint-space)
													// movej(q, a=1.4, v=1.05, t=0, r =0)
		q1 := DEG_TO_RAD(Prozessvariablen.q1);
		q2 := DEG_TO_RAD(Prozessvariablen.q2);
		q3 := DEG_TO_RAD(Prozessvariablen.q3);
		q4 := DEG_TO_RAD(Prozessvariablen.q4);
		q5 := DEG_TO_RAD(Prozessvariablen.q5);
		q6 := DEG_TO_RAD(Prozessvariablen.q6);
		
		stringFormat(sFormat := 'movej([%.3f,%.3f,%.3f,%.3f,%.3f,%.3f], a=%.2f, v=%.2f)',
							arg1 := F_LREAL(q1),
							arg2 := F_LREAL(q2),
							arg3 := F_LREAL(q3),
							arg4 := F_LREAL(q4),
							arg5 := F_LREAL(q5),
							arg6 := F_LREAL(q6),
							arg7 := F_LREAL(Prozessvariablen.a),
							arg8 := F_LREAL(Prozessvariablen.v),
							bError => bFehler,
							nErrId => iErrorID,
							sOut => Command);	
													
	END_IF
	
	IF Prozessvariablen.MoveTyp = 2 THEN			// Move Circular: Move to position (circular in tool-space)
													//movec(pose_via, pose_to, a=1.2, v=0.25, r =0, mode=0)
													
		
	END_IF
	
	IF Prozessvariablen.MoveTyp = 3 THEN			// Move Process
													// movep(pose, a=1.2, v=0.25, r=0)
		stringFormat(sFormat := 'movep(%s, a=%.2f, v=%.2f)',
							arg1 := F_STRING(pose),
							arg2 := F_LREAL(Prozessvariablen.a),
							arg3 := F_LREAL(Prozessvariablen.v),
							bError => bFehler,
							nErrId => iErrorID,
							sOut => Command);												
	END_IF

// Vorbereiten von Array
	CommandArray.sValue := Command;
	CommandArray.arrByte[LEN(CommandArray.sValue)] := 10;

// Senden von Array	
	Send_START(cbLen := LEN(CommandArray.sValue),
			pSrc := ADR(CommandArray.arrByte),
			bExecute := TRUE);
	GVL.ObjectArray[GVL.CountObject] := CommandArray.sValue;
			
	GVL.CountObject := GVL.CountObject + 1;
			
	IF NOT Send_START.bBusy THEN
		Send_START(bExecute := FALSE);
		M_BewegungZuPosition := TRUE;
	END_IF
END_METHOD

METHOD M_Reset : BOOL
bResettenSkill := TRUE;

IF bResettenSkill THEN
	M_Reset := TRUE;
ELSE
	M_Reset := FALSE;
END_IF
END_METHOD

METHOD M_Start : BOOL
GVL.CountObjectStart := GVL.CountObjectStart + 1;

// Prüfen von Bedingungen
	// Ist das  System im korrekten Status
	IF eSysState = 1 OR eSysState = 2 THEN
		// Ist das Objekt im korrekten Status 
		IF iState = 1 THEN
			bResettenSkill := FALSE;
			bStarten := TRUE;
		END_IF
	END_IF

IF bStarten THEN
	M_Start := TRUE;
ELSE
	M_Start := FALSE;
END_IF
END_METHOD

METHOD M_Stop : BOOL
// Ist das Objekt im korrekten Status 
	IF iState = 3 THEN
		bSkillFertig := TRUE;
	END_IF

IF bSkillFertig THEN
	M_Stop := TRUE;
ELSE
	M_Stop := FALSE;
END_IF
END_METHOD

METHOD M_Trennen : BOOL
VAR_INPUT
END_VAR
// Ausführen von Funktionalitäten
	Disconnect(sSrvNetId := sSrvNetId,
			bExecute := TRUE,
			tTimeout := tTimeout,
			bError => bFehler,
			nErrId => iErrorID);
	
	IF NOT Disconnect.bBusy AND NOT bFehler THEN
		M_Trennen := TRUE;
		Disconnect(bExecute := FALSE);
	END_IF
END_METHOD

METHOD M_Verbinden : BOOL 
VAR
	
END_VAR
// Ausführen von Funktionalitäten
	Connect(sSrvNetId := sSrvNetId,
			sRemoteHost := sIP,
			nRemotePort := iPort_Prim,
			bExecute := TRUE,
			tTimeout := tTimeout,
			bError => bFehler,
			nErrId => iErrorID,
			hSocket => hSocket);
			
	IF hSocket.handle <> 0 THEN
		M_Verbinden := TRUE;
		Connect(bExecute := FALSE);
		Connect_RT(bExecute := FALSE);
	END_IF
END_METHOD

PROPERTY P_Prozessparameter : sRoboterProzessVariablen
SET
Prozessvariablen := P_Prozessparameter;
END_SET
END_PROPERTY

PROPERTY P_State : eObjectAktorState
GET
P_State := iState;
END_GET
END_PROPERTY

PROPERTY Test_Param : sRoboterProzessVariablen
GET
Test_Param := Prozessvariablen;
END_GET
END_PROPERTY

END_FUNCTION_BLOCK

// ---- POUs/02_Anlagenmodell/01_Objektklassen/00_Referenz/FB_Basis_Objekt_Aktor.TcPOU
FUNCTION_BLOCK FB_Basis_Objekt_Aktor
VAR_INPUT
	// Betriebsvariablen
	eSysState				:eSystemState;			// Information über Stand von System
	eSysCommand		  		:eSystemCommand;		// Steuerungsvariabel von System
	iMode					:INT;					// Information über aktuellen Betriebsmodi 
END_VAR
VAR_OUTPUT
	iErrorID				:UDINT;					// Information um welchen Fehler es sich handelt	
END_VAR
VAR
	// Managementvariablen
	iState					:eObjectAktorState;		// Information über Zustand von Objekt
	
	// Zustandsvariablen
	bEinschalten			:BOOL;				// Objekt einschalten
	bAusschalten			:BOOL;				// Objekt ausschalten
 	bStarten				:BOOL;				// Objekt starten
	bObjektFertig			:BOOL;				// Objekt hat Prozess abgeschlossen
	bSkillFertig			:BOOL;				// Skill hat Prozess abgeschlossen
	bStoppen				:BOOL;				// Objekt wurde gestoppt
	bResettenSkill			:BOOL;				// Das Objekt wird durch den Skill resettet
	bResettenSystem			:BOOL;				// Das Objekt wird durch das System resettet 
	bFehler					:BOOL;				// Das Objket hat einen Fehler
END_VAR

END_FUNCTION_BLOCK

// ---- POUs/02_Anlagenmodell/01_Objektklassen/FB_SmartGreifer.TcPOU
FUNCTION_BLOCK FB_SmartGreifer IMPLEMENTS I_Objekt_SmartGreifer
VAR_INPUT
	eSysState			:eSystemState;		// Information über Stand von System
	eSysCommand		  	:eSystemCommand;	// Steuerungsvariabel von System
	iMode				:INT;				// Information über aktuellen Betriebsmodi 
END_VAR
VAR_OUTPUT
	iErrorID			:UDINT;				// Information um welchen Fehler es sich handelt	
END_VAR
VAR
	
	iState				:eObjectAktorState;		// Information über Zustand von Skill
	
	// Zustandsvariablen
	bEinschalten			:BOOL;			// Objekt einschalten
	bAusschalten			:BOOL;			// Objekt ausschalten
 	bStarten				:BOOL;			// Objekt starten
	bObjektFertig			:BOOL;			// Objekt hat Prozess abgeschlossen
	bSkillFertig			:BOOL;			// Skill hat Prozess abgeschlossen
	bStoppen				:BOOL;			// Objekt wurde gestoppt
	bResettenSkill			:BOOL;			// Das Objekt wird durch den Skill resettet
	bResettenSystem			:BOOL;			// Das Objekt wird durch das System resettet 
	bFehler					:BOOL;			// Das Objket hat einen Fehler
	
	iFehlerID				:UDINT;


	// Instanziierung von Kommunikationsbausteine 
	Communication			:ModbusRtuMasterV2_KL6x22B;
	
	// Kommunikationsvariablen
	UnitID      			:BYTE := 9;
    Quantity    			:WORD;
    MBAddr      			:WORD;
	Timeout     			:TIME := T#5S;
	cbRead					:UINT;
	DataSend				:ARRAY[0..5] OF BYTE;
	DataRead				:ARRAY[0..5] OF BYTE;
	
	// Managementvariablen
	iStartUp			:INT;
	iProzess			:INT;
	
	bGreiferReset		:BOOL;
	bGreiferLesen		:BOOL;
	
	bAmEinschalten		:BOOL;
	bEingeschalten		:BOOL;
	
	bGestartet			:BOOL;
	
	
	CheckTimer			:TON;
	Delay				:TON;
	
	// Prozessvariablen
	iPos				:BYTE;
	iGeschw				:BYTE;
	iKraft				:BYTE;
	
	// Eigenschaftsvariablen
	iPosMax				:REAL := 85;
	iGeschwMin			:REAL := 20;
	iGeschwMax			:REAL := 150;
	iKraftMin			:REAL := 20;
	iKraftMax			:REAL := 235;
	Anschlag			:BYTE;
	Prozessvariablen 	:sSmartGreiferProzessVariablen;

	TestCheck			:BOOL;
	
	
END_VAR

// Instanziierungen	
Communication(
	UnitID 		:= UnitID,
	Timeout 	:= Timeout,
	Error 		=> bFehler,
	ErrorId 	=> iErrorID,
	cbRead 		=> cbRead);


//____________________________________________________________________________________________
// Input-Command-Verwaltung
	// System
	IF eSysCommand = 2 AND iState = 0 THEN			// Objekt einschalten
		bEinschalten := TRUE;
	ELSE 
		bEinschalten := FALSE;
	END_IF
	
	IF eSysCommand = 1 AND iState = 1 THEN				// Objekt ausschalten
		bAusschalten := TRUE;		
	ELSE 
		bAusschalten := FALSE;		
	END_IF
	
	IF eSysCommand = 3 THEN								// Objekt beendet Prozess
		bStoppen := TRUE;
	ELSE
		bStoppen := FALSE;
	END_IF
	
	IF eSysCommand = 4 THEN								// System resettet Objekt
		bResettenSystem := TRUE;
	ELSE
		bResettenSystem := FALSE;
	END_IF

//____________________________________________________________________________________________
// Interner Methodenaufruf (Durch System oder Skill)

//____________________________________________________________________________________________
// Datenerfassungsprozess

//____________________________________________________________________________________________
// Zustandsmanagement

IF bFehler THEN 
	iState := 7;
END_IF

CASE iState OF 
	0: // AUS
		// DO
		IF bEinschalten THEN
			CASE iStartUP OF
				0: // Greifer Resetten
					bGreiferReset := M_Resetten();
					
					IF bGreiferReset THEN
						bGreiferReset := FALSE;
						iStartUp := 1;
					END_IF
				1: // Greifer Aktivieren
					bAmEinschalten := M_Aktivieren();
					
					IF bAmEinschalten THEN 
						bAmEinschalten := FALSE;
						Delay(IN:= TRUE, PT := T#1S);
					END_IF
					
					IF Delay.Q THEN
						Delay(IN:= FALSE);
						iStartUp := 2;
					END_IF
					
				2:
					bGreiferLesen := M_StatusLesen(NrOfReg := 1);
					
					IF bGreiferLesen THEN
						bGreiferLesen := FALSE;
						IF DataRead[1] = 49  AND DataRead[0] = 0 THEN
							bEingeschalten := TRUE;
						END_IF
					END_IF
			END_CASE
		END_IF
		
		// TRANSITION
		IF bEingeschalten THEN																			// Verbindung wird aufgebaut
			bEingeschalten := FALSE;
			iStartUp := 0;
			iState := 1;
		END_IF
			
	//____________________________________________________________________________________________
	1: // BEREIT
		// DO
			Anschlag := 0;

		// TRANSITION		
			IF bAusschalten THEN
				iState := 0;
			END_IF
																									// Manuell-Modus wird eingeschalten
													
			 IF bStarten THEN																		// Objekt führt Prozessdurch
				 bStarten := FALSE;
				 iState := 3;
			 END_IF			
	//____________________________________________________________________________________________
	2: // MANUELL
		// DO
		
		// TRANSITION
	
	//____________________________________________________________________________________________
	3: // LAUFEND
		// DO
			
			// Aktionsprozess 
				CASE iProzess OF 
				0: // Aktion durchführen
					iPos := REAL_TO_BYTE((255.00/iPosMax) *  (iPosMax - Prozessvariablen.Pos));	
					iGeschw := REAL_TO_BYTE((255.00 / 100.00) * Prozessvariablen.Geschw );
					iKraft := REAL_TO_BYTE((255.00 / 100.00) * Prozessvariablen.F);
				
					bGestartet := M_PositionAnfahren(iPos := iPos, iGeschw := iGeschw, iKraft := iKraft);
					
					IF bGestartet THEN
						bGestartet := FALSE;
						Delay(IN:= TRUE, PT := T#1S);
					END_IF
					
					IF Delay.Q THEN
						Delay(IN:= FALSE);
						iProzess := 1;
					END_IF
				
				1: // Prüfen ob Aktion erledigt 
					bGreiferLesen := M_StatusLesen(NrOfReg := 3);
					CheckTimer(IN := TRUE, PT := T#5S);
					
					IF bGreiferLesen THEN
						bGreiferLesen := FALSE;
						
						// Greifer hat Position erreicht
						IF 	DataRead[0] = 0 		AND
							DataRead[1] = 249 		AND
							DataRead[2] = iPos 		AND
							DataRead[3] = 0 		AND
							DataRead[4] = 0 		AND
							DataRead[5] = iPos		THEN
							
							CheckTimer(IN := FALSE);
							iProzess := 0;
							bObjektFertig := TRUE;
						END_IF
						
						// Greifer ist in Hinderniss gefahren
						IF 	DataRead[0] = 0 		AND
							//DataRead[1] = 185 		AND
							DataRead[2] = iPos 		AND
							DataRead[3] = 0 		AND
							DataRead[4] <> 0 		THEN
							
							Anschlag := DataRead[5];
							CheckTimer(IN := FALSE);
							iProzess := 0;
							bObjektFertig := TRUE;
						END_IF
						
					END_IF
					
					// Zeit wurde überschritten
					IF CheckTimer.Q THEN		
						iProzess := 0;
						CheckTimer(IN := FALSE);
						bFehler := TRUE;
						iFehlerID := 201;
					END_IF
				END_CASE
						
		// TRANSITION
			IF bObjektFertig THEN
				bObjektFertig := FALSE;
				iState := 4;
				TestCheck := TRUE;
			END_IF
			
			IF bSkillFertig THEN
				bSkillFertig := FALSE;
				iState := 5;
			END_IF
				
			IF bStoppen THEN
				iState := 6;
			END_IF
					
	
	//____________________________________________________________________________________________
	4: // ABGESCHLOSSEN_INTERN
		// DO
		TestCheck := FALSE;
		// TRANSITION
			IF bResettenSkill THEN																	// Objekt resetten
				bResettenSkill := FALSE;		
				iState := 1;
			END_IF
	//____________________________________________________________________________________________
	5: // ABGESCHLOSSEN_EXTERN
		// DO																					
		
		// TRANSITION
			IF bResettenSkill THEN																	// Objekt resetten
				bResettenSkill := FALSE;
				iState := 1;
			END_IF
	
	//____________________________________________________________________________________________
	6: // GESTOPPT
		// DO
		
		// TRANSITION
			IF bResettenSystem THEN																	// Objekt resetten
				iState := 1;
			END_IF
	
	//____________________________________________________________________________________________
	7: // FEHLER
		// DO
			iErrorID := iFehlerID;
			
		// TRANSITION
			IF bResettenSystem THEN																	// Objekt resetten
				bFehler	 := FALSE;
				iErrorID := 0;
				iState := 1;
			END_IF
	
END_CASE

METHOD M_Aktivieren : BOOL
VAR_INPUT
END_VAR
// Definieren der Anzahl von Daten-Bytes 
Quantity := 3;

// Definieren von Register
MBAddr := 1000;

// Definieren der Daten
DataSend[0] := 0;
DataSend[1] := 1;
DataSend[2] := 0;
DataSend[3] := 0;
DataSend[4] := 0;
DataSend[5] := 0;

// Senden von Daten an entsprechendes Register
Communication.WriteRegs(
	Quantity 	:= Quantity,
	MBAddr 		:= MBAddr,
	cbLength 	:= SIZEOF(DataSend),
	pMemoryAddr := ADR(DataSend),
	Execute 	:= TRUE);
	
IF NOT Communication.BUSY THEN
	Communication.WriteRegs(Execute := FALSE);
	M_Aktivieren := TRUE;
END_IF
END_METHOD

METHOD M_PositionAnfahren : BOOL
VAR_INPUT
	iPos		:BYTE;
	iGeschw		:BYTE;
	iKraft		:BYTE;
END_VAR

// Definieren der Anzahl von Daten-Bytes 
Quantity := 3;

// Definieren von Register
MBAddr := 1000;

// Definieren der Daten
DataSend[0] := 0;
DataSend[1] := 9;
DataSend[2] := iPos;
DataSend[3] := 0;
DataSend[4] := iKraft;
DataSend[5] := iGeschw;

// Senden von Daten an entsprechendes Register
Communication.WriteRegs(
	Quantity 	:= Quantity,
	MBAddr 		:= MBAddr,
	cbLength 	:= SIZEOF(DataSend),
	pMemoryAddr := ADR(DataSend),
	Execute 	:= TRUE);
	
IF NOT Communication.BUSY THEN
	Communication.WriteRegs(Execute := FALSE);
	M_PositionAnfahren := TRUE;
END_IF
END_METHOD

METHOD M_Reset : BOOL
bResettenSkill := TRUE;

IF bResettenSkill THEN
	M_Reset := TRUE;
ELSE
	M_Reset := FALSE;
END_IF
END_METHOD

METHOD M_Resetten : BOOL
VAR_INPUT
END_VAR
// Definieren der Anzahl von Daten-Bytes 
Quantity := 3;

// Definieren von Register
MBAddr := 1000;

// Definieren der Daten
DataSend[0] := 0;
DataSend[1] := 0;
DataSend[2] := 0;
DataSend[3] := 0;
DataSend[4] := 0;
DataSend[5] := 0;

// Senden von Daten an entsprechendes Register
Communication.WriteRegs(
	Quantity 	:= Quantity,
	MBAddr 		:= MBAddr,
	cbLength 	:= SIZEOF(DataSend),
	pMemoryAddr := ADR(DataSend),
	Execute 	:= TRUE);
	
IF NOT Communication.BUSY THEN
	Communication.WriteRegs(Execute := FALSE);
	M_Resetten := TRUE;
END_IF
END_METHOD

METHOD M_Start : BOOL
// Prüfen von Bedingungen
	// Ist das  System im korrekten Status
	IF eSysState = 1 OR eSysState = 2 THEN
		// Ist das Objekt im korrekten Status 
		IF iState = 1 THEN
			// Prüfen auf Fehler (Muss ergänzt werden)
				bResettenSkill := FALSE;
				bStarten := TRUE;
		END_IF
	END_IF

IF bStarten THEN
	M_Start := TRUE;
ELSE
	M_Start := FALSE;
END_IF
END_METHOD

METHOD M_StatusLesen : BOOL
VAR_INPUT
	NrOfReg			:WORD;
END_VAR
// Definieren von Register
MBAddr := 2000;


// Lesen von Daten des entsprechenden Registers
Communication.ReadRegs(
	Quantity 	:= NrOfReg,
	MBAddr 		:= MBAddr,
	cbLength 	:= SIZEOF(DataRead),
	pMemoryAddr := ADR(DataRead),
	Execute 	:= TRUE);
	
	
IF NOT Communication.BUSY THEN
	Communication.ReadRegs(Execute := FALSE);
	M_StatusLesen := TRUE;
END_IF
END_METHOD

METHOD M_Stop : BOOL
// Ist das Objekt im korrekten Status 
	IF iState = 3 THEN
		bStoppen := TRUE;
	END_IF

IF bStoppen THEN
	M_Stop := TRUE;
ELSE
	M_Stop := FALSE;
END_IF
END_METHOD

PROPERTY P_AnschlagPos : BYTE
GET
P_AnschlagPos := Anschlag;
END_GET
END_PROPERTY

PROPERTY P_Prozessparameter : sSmartGreiferProzessVariablen
SET
Prozessvariablen := P_Prozessparameter;
END_SET
END_PROPERTY

PROPERTY P_State : eObjectAktorState
GET
P_State := iState;
END_GET
END_PROPERTY

END_FUNCTION_BLOCK

// ---- POUs/02_Anlagenmodell/01_Objektklassen/FB_Kraftsensor_V2.TcPOU
FUNCTION_BLOCK FB_Kraftsensor_V2 IMPLEMENTS I_Objekt_Kraftsensor
VAR_INPUT
	eSysState			:eSystemState;		// Information über Stand von System
	eSysCommand		  	:eSystemCommand;	// Steuerungsvariabel von System
	iMode				:INT;				// Information über aktuellen Betriebsmodi 
	
	// Kommunikationsvariablen
	sIP					:T_IPv4Addr;
	iPort				:UINT;
END_VAR
VAR_OUTPUT
	iErrorID			:UDINT;					// Information um welchen Fehler es sich handelt	
END_VAR
VAR
	iState				:eObjectSensorState;	// Information über Zustand von Skill
	
	// Zustandsvariablen
	bEinschalten			:BOOL;			// Objekt einschalten
	bAusschalten			:BOOL;			// Objekt ausschalten
	bResettenSystem			:BOOL;			// Das Objekt wird durch das System resettet 
	bFehler					:BOOL;			// Das Objket hat einen Fehler
	
	iFehlerID				:UDINT;


	// Instanziierung von Kommunikationsbausteine
	Connect				:FB_SocketConnect;
	Disconnect			:FB_SocketClose;
	Send				:FB_SocketSend;
	Receive				:FB_SocketReceive;
	
	// Kommunikationsvariablen
	sSrvNetId   		:T_AmsNetId := '';
	tTimeout    		:TIME := T#45S;(*!!!*)
	hSocket    			:T_HSOCKET;
	
	// RealTimeDatenerfassung
	RT_State			:INT;							// RealTime-State-Variable
	{attribute 'TcSwapWord'}
	SendData 			:Request;
	{attribute 'TcSwapWord'}
	ReceivedData		:Response_Values;				// Erhaltene Daten von Roboter
	nRecBytes			:UDINT;							// Anzahl der erhaltenen Bytes
	
	CPF					:INT := 10000;					// Counts per Force value
	CPT					:INT := 10000;					// Counts per Torque value (Noch mal 10 rechnen)
	ScalefactorFx		:INT := 200;					// Additional scaling factor (for the Fx,Fy,Fz,Tx,Ty,Tz)
	ScalefactorFy		:INT := 200;					// Additional scaling factor (for the Fx,Fy,Fz,Tx,Ty,Tz)
	ScalefactorFz		:INT := 200;					// Additional scaling factor (for the Fx,Fy,Fz,Tx,Ty,Tz)
	ScalefactorTx		:INT := 100;					// Additional scaling factor (for the Fx,Fy,Fz,Tx,Ty,Tz)
	ScalefactorTy		:INT := 100;					// Additional scaling factor (for the Fx,Fy,Fz,Tx,Ty,Tz)
	ScalefactorTz		:INT := 65;						// Additional scaling factor (for the Fx,Fy,Fz,Tx,Ty,Tz)
	
	RohArray			:Int_2Byte;
	SwitchArray			:ARRAY[0..1] OF BYTE;
	SwichValue			:Array2_Int;
		
	Rohdaten			:Kraftvariablen;				// Rohwerte der Messung 
	Messung				:Kraftvariablen;				// Werte in Newton / Newtonmeter 

	// Managementvariablen
	bAusgeschalten		:BOOL;
	bManOn				:BOOL;
	m					:INT;
	
	// Eigenschaftsmethoden
	sLimitGrenze		:sKraftVariablen;
	sErreichtGrenze		:sKraftVariablen;
	bLimit				:BOOL;
	bLimitx				:BOOL;
	bLimity				:BOOL;
	bLimitz				:BOOL;
	bErreicht			:BOOL;
	bErreichtx			:BOOL;
	bErreichty			:BOOL;
	bErreichtz			:BOOL;
	
END_VAR

// Instanziierungen
Connect(sSrvNetId := sSrvNetId,
		sRemoteHost := sIP,
		nRemotePort := iPort,
		tTimeout := tTimeout,
		bError => bFehler,
		nErrId => iErrorID,
		hSocket => hSocket);	
						
Send(sSrvNetId := sSrvNetId,
		hSocket := hSocket,
		tTimeout := tTimeout,
		cbLen := SIZEOF(SendData),
		pSrc := ADR(SendData),
		bError => bFehler,
		nErrId => iErrorID);
						
Receive(sSrvNetId := sSrvNetId,
		hSocket := hSocket,
		cbLen := SIZEOF(ReceivedData),
		pDest := ADR(ReceivedData),
		tTimeout := tTimeout,
		bError => bFehler,
		nErrId => iErrorID,
		nRecBytes => nRecBytes);
						
Disconnect(sSrvNetId := sSrvNetId,
			hSocket := hSocket,
			tTimeout := tTimeout,
			bError => bFehler,
			nErrId => iErrorID);

//____________________________________________________________________________________________
// Input-Command-Verwaltung
IF eSysCommand = 2 AND iState = 0 THEN				// Objekt einschalten
		bEinschalten := TRUE;
	ELSE 
		bEinschalten := FALSE;
	END_IF
	
	IF eSysCommand = 1 AND iState = 1 THEN			// Objekt ausschalten
		bAusschalten := TRUE;		
	ELSE 
		bAusschalten := FALSE;		
	END_IF
	
	IF eSysCommand = 4 THEN							// System resettet Objekt
		bResettenSystem := TRUE;
	ELSE
		bResettenSystem := FALSE;
	END_IF

//____________________________________________________________________________________________
// Interner Methodenaufruf (Durch System oder Skill)

//____________________________________________________________________________________________
// Datenerfassungsprozess
IF bManOn OR iState = 1 THEN
	CASE RT_State OF 
		0:	// Connect to RealTimePort
				Connect(bExecute := TRUE);			
					
				IF NOT Connect.bBusy AND NOT Connect.bError THEN
					Connect.bExecute := FALSE;
					RT_State := 1;
				END_IF
				
		1: 	// Send Data 
					SendData.Command := 0;
					Send(bExecute := TRUE);
				
					IF NOT Send.bBusy AND NOT Send.bError THEN
						Send.bExecute := FALSE;
						RT_State := 2;
					END_IF
		
		2:	// Get Data 
				Receive(bExecute := TRUE);
			
				IF NOT Receive.bBusy AND NOT Receive.bError THEN
					Receive.bExecute := FALSE;
					RT_State := 3;
				END_IF
				
		3:	// Convert Data
		
			RohArray.sValue := ReceivedData.Fx;
			SwitchArray[0] := RohArray.arrByte[1];
			SwitchArray[1] := RohArray.arrByte[0];
			SwichValue.arrByte := SwitchArray;
			Rohdaten.Fx := SwichValue.sValue;
			Messung.Fx := Rohdaten.Fx * ScalefactorFx / (CPF);
			
			RohArray.sValue := ReceivedData.Fy;
			SwitchArray[0] := RohArray.arrByte[1];
			SwitchArray[1] := RohArray.arrByte[0];
			SwichValue.arrByte := SwitchArray;
			Rohdaten.Fy := SwichValue.sValue;
			Messung.Fy := Rohdaten.Fy * ScalefactorFy / (CPF);
			
			RohArray.sValue := ReceivedData.Fz;
			SwitchArray[0] := RohArray.arrByte[1];
			SwitchArray[1] := RohArray.arrByte[0];
			SwichValue.arrByte := SwitchArray;
			Rohdaten.Fz := SwichValue.sValue;
			Messung.Fz := Rohdaten.Fz * ScalefactorFz / (CPF);
			
			RohArray.sValue := ReceivedData.Tx;
			SwitchArray[0] := RohArray.arrByte[1];
			SwitchArray[1] := RohArray.arrByte[0];
			SwichValue.arrByte := SwitchArray;
			Rohdaten.Tx := SwichValue.sValue;
			Messung.Tx := Rohdaten.Tx * ScalefactorTx / (CPT);
			
			RohArray.sValue := ReceivedData.Ty;
			SwitchArray[0] := RohArray.arrByte[1];
			SwitchArray[1] := RohArray.arrByte[0];
			SwichValue.arrByte := SwitchArray;
			Rohdaten.Ty := SwichValue.sValue;
			Messung.Ty := Rohdaten.Ty * ScalefactorTy / (CPT);
			
			RohArray.sValue := ReceivedData.Tz;
			SwitchArray[0] := RohArray.arrByte[1];
			SwitchArray[1] := RohArray.arrByte[0];
			SwichValue.arrByte := SwitchArray;
			Rohdaten.Tz := SwichValue.sValue;
			Messung.Tz := Rohdaten.Tz * ScalefactorTz / (CPT);
			
		
			RT_State := 4;
				
		4:	// Disconnect from RealTimePort
				Disconnect(bExecute := TRUE);
							
				IF NOT Disconnect.bBusy AND NOT Disconnect.bError THEN
					Disconnect.bExecute := FALSE;
					RT_State := 0;
				END_IF
	END_CASE
END_IF

//____________________________________________________________________________________________
// Zustandsmanagement
IF bFehler THEN 
	iState := 2;
END_IF

CASE iState OF 
	0: // AUS
		// DO
			RT_State := 0;
			
			Messung.Fx := 0;
			Messung.Fy := 0;
			Messung.Fz := 0;
			Messung.Tx := 0;
			Messung.Ty := 0;
			Messung.Tz := 0;
		
		// TRANSITION	
			IF bEinschalten THEN																	// Verbindung wird aufgebaut
				iState := 1;
			END_IF
			
	//____________________________________________________________________________________________
	1: // LAUFEND
		// DO
			IF bAusschalten THEN																	// Objekt ausschalten	
				Disconnect(bExecute := TRUE);
				IF NOT Disconnect.bBusy AND NOT Disconnect.bError THEN
					Disconnect.bExecute := FALSE;
					bAusgeschalten := TRUE;
				END_IF	
			END_IF
		
		// TRANSITION
			IF bAusgeschalten THEN																	// Objekt ausschalten
				bAusgeschalten := FALSE;
				iState := 0;
			END_IF
	
	//____________________________________________________________________________________________
	2: // FEHLER
		// DO
		
		// TRANSITION
		IF bResettenSystem THEN																	// Objekt resetten
			bFehler	 := FALSE;
			iState := 1;
		END_IF
	
END_CASE

PROPERTY P_Messdaten : Kraftvariablen
GET
P_Messdaten := Messung;
END_GET
END_PROPERTY

PROPERTY P_State : eObjectSensorState
GET
END_GET
END_PROPERTY

END_FUNCTION_BLOCK

// ---- POUs/03_Systemmodell/Systemparameter.TcPOU
PROGRAM Systemparameter
VAR
END_VAR

// Lesen
	// Objektzustände
	GVL.Robot_State 		:= Anlage.UR5.P_State;
	GVL.Greifer_State 		:= Anlage.Gripper.P_State;
	GVL.Sensor_State 		:= 1;

// Zuweisen
	// Eigenschaften

END_PROGRAM

// ---- POUs/03_Systemmodell/Zustandshandling.TcPOU
PROGRAM Zustandshandling
VAR
	iState			:eSystemState;
	
	bEinschalten	:BOOL;
	bAusschalten	:BOOL;
	bStarten		:BOOL;
	bStoppen		:BOOL;
	bFehler			:BOOL;
	bResetten		:BOOL;
	bAbgeschlossen	:BOOL;
END_VAR

GVL.SystemState := iState;

CASE iState OF
	0:	// AUS
			// DO
			IF GVL.Greifer_State = 1 AND GVL.Robot_State = 1 AND GVL.Sensor_State = 1 THEN
				bEinschalten := TRUE;
			END_IF
			
			// TRANSITION
			IF bEinschalten THEN
				bEinschalten := FALSE;
				iState := 1;
			END_IF
		
			
	1:	// BEREIT
			// DO
			IF GVL.Greifer_State = 3 AND GVL.Robot_State = 3 AND GVL.Sensor_State = 3 THEN
				bStarten := TRUE;
			END_IF
			
			IF GVL.Greifer_State = 0 THEN
				bAusschalten := TRUE;
			END_IF
			
			IF GVL.ErrorID <> 0 THEN
				bFehler := TRUE;
			END_IF
			
			// TRANSITION
			IF bStarten THEN
				bStarten := FALSE;
				iState := 2;
			END_IF
			
			IF bAusschalten THEN
				bAusschalten := FALSE; 
				iState := 0;
			END_IF
			
			IF bFehler THEN
				bFehler := FALSE;
				iState := 4;
			END_IF
			
	2:	// LAUFEND
			// DO
			IF GVL.SystemCommand = 3 THEN
				bStoppen := TRUE;
			END_IF
			
			IF GVL.Greifer_State = 1 AND GVL.Robot_State = 1 AND GVL.Sensor_State = 1  THEN
				bAbgeschlossen := TRUE;
			END_IF
			
			IF GVL.ErrorID <> 0 THEN
				bFehler := TRUE;
			END_IF
			
			// TRANSITION
			IF bStoppen THEN
				bStoppen := FALSE;
				iState := 3;
			END_IF
			
			IF bAbgeschlossen THEN
				bAbgeschlossen := FALSE;
				iState := 1;
			END_IF
			
			IF bFehler THEN
				bFehler := FALSE;
				iState := 4;
			END_IF
			
	3:	// GESTOPPT
			// DO
			IF GVL.SystemCommand = 4 THEN
				bResetten := TRUE;
			END_IF
			
			// TRANSITION
			IF bResetten THEN
				bResetten := FALSE;
				iState := 1;
			END_IF
			
	4:	// FEHLER
			// DO
			IF GVL.SystemCommand = 4 THEN
				bResetten := TRUE;
			END_IF
			
			// TRANSITION
			IF bResetten THEN
				bResetten := FALSE;
				iState := 1;
			END_IF
			
END_CASE

END_PROGRAM

// ---- POUs/PunkteZuweisung_Temp.TcPOU
PROGRAM PunkteZuweisung_Temp
VAR
	// Roboterpositionen
		// Fixe Postionene
		PHome				:sRoboterProzessVariablen;
		PGetPlate1			:sRoboterProzessVariablen;
		PGetPlate2			:sRoboterProzessVariablen;
		PStartSetPlate1		:sRoboterProzessVariablen;
		PStartSetPlate2		:sRoboterProzessVariablen;
		PStartAPlate		:sRoboterProzessVariablen;
		PStartAXFixPlate	:sRoboterProzessVariablen;
		PStartAYFixPlate	:sRoboterProzessVariablen;
		PGetFixPlate		:sRoboterProzessVariablen;
		PStartSetFixPlate	:sRoboterProzessVariablen;
		
		
		// Offsets
		POffsetZ		:sRoboterProzessVariablen;
		POffsetnZ		:sRoboterProzessVariablen;
		POffsetXs		:sRoboterProzessVariablen;
		POffsetnXs		:sRoboterProzessVariablen;
		POffsetnYs		:sRoboterProzessVariablen;
		
		// Ausrichtungs_Offsets
		POffsetAX		:sRoboterProzessVariablen;
		POffsetAnX		:sRoboterProzessVariablen;
		POffsetAY		:sRoboterProzessVariablen;
		POffsetAnY		:sRoboterProzessVariablen;
		POffsetAnZ		:sRoboterProzessVariablen;
	
	// Greiferpositionen		
		Plate_Open		:sSmartGreiferProzessVariablen;
		Plate_Closed	:sSmartGreiferProzessVariablen;
		FixPlate_Open	:sSmartGreiferProzessVariablen;
		FixPlate_Closed	:sSmartGreiferProzessVariablen;
		GripperClossed	:sSmartGreiferProzessVariablen;
	
	// Kraftvariablen
	AnstossX		:sKraftVariablen;
	AnstossnX		:sKraftVariablen;
	AnstossY		:sKraftVariablen;
	AnstossnY		:sKraftVariablen;
	AnstossZ		:sKraftVariablen;
	
	// Datenpakete
	R_Data_1				:ARRAY[0..2] OF sRoboterProzessVariablen;	
	R_Data_2				:ARRAY[0..4] OF sRoboterProzessVariablen;
	R_Data_3				:ARRAY[0..2] OF sRoboterProzessVariablen;
	R_Data_4				:ARRAY[0..3] OF sRoboterProzessVariablen;
	R_Data_5				:ARRAY[0..4] OF sRoboterProzessVariablen;
	R_Data_6				:ARRAY[0..4] OF sRoboterProzessVariablen;
	R_Data_7				:ARRAY[0..4] OF sRoboterProzessVariablen;
	R_Data_8				:ARRAY[0..2] OF sRoboterProzessVariablen;
	R_Data_9				:ARRAY[0..2] OF sRoboterProzessVariablen;
	
	G_Data_1				:ARRAY[0..1] OF sSmartGreiferProzessVariablen;
	G_Data_2				:ARRAY[0..1] OF sSmartGreiferProzessVariablen;
	
	S_Data_1				:ARRAY[0..1] OF sKraftVariablen;
	
	
END_VAR

// Roboterpositionen
	// Fixe Positionen
		// Homeposition
		pHome.q1 := 90;
		pHome.q2 := -90;
		pHome.q3 := -90;
		pHome.q4 := -90;
		pHome.q5 := 90;
		pHome.q6 := 180;
		pHome.v := 0.5;
		pHome.a := 0.5;
		pHome.MoveTyp := 1;
		pHome.PosTyp := 0;
		
		// Lagerposition von Platte 1
		PGetPlate1.q1 := 0.070;
		PGetPlate1.q2 := 0.583;
		PGetPlate1.q3 := 0.236;
		PGetPlate1.q4 := 0;
		PGetPlate1.q5 := -180;
		PGetPlate1.q6 := 0;
		PGetPlate1.v := 1;
		PGetPlate1.a := 1;
		PGetPlate1.MoveTyp := 3;
		PGetPlate1.PosTyp := 0;
		
		// Lagerposition von Platte 2
		PGetPlate2.q1 := 0.166;
		PGetPlate2.q2 := 0.583;
		PGetPlate2.q3 := 0.236;
		PGetPlate2.q4 := 0;
		PGetPlate2.q5 := -180;
		PGetPlate2.q6 := 0;
		PGetPlate2.v := 1;
		PGetPlate2.a := 1;
		PGetPlate2.MoveTyp := 3;
		PGetPlate2.PosTyp := 0;
		
		// Startposition für Platzierung von Platte 1
		PStartSetPlate1.q1 := 0.070;
		PStartSetPlate1.q2 := 0.490;
		PStartSetPlate1.q3 := 0.236;
		PStartSetPlate1.q4 := 0;
		PStartSetPlate1.q5 := -180;
		PStartSetPlate1.q6 := 0;
		PStartSetPlate1.v := 1;
		PStartSetPlate1.a := 1;
		PStartSetPlate1.MoveTyp := 3;
		PStartSetPlate1.PosTyp := 0;
		
		// Startposition für Platzierung von Platte 2
		PStartSetPlate2.q1 := 0.165;
		PStartSetPlate2.q2 := 0.471;
		PStartSetPlate2.q3 := 0.236;
		PStartSetPlate2.q4 := 0;
		PStartSetPlate2.q5 := -180;
		PStartSetPlate2.q6 := 0;
		PStartSetPlate2.v := 1;
		PStartSetPlate2.a := 1;
		PStartSetPlate2.MoveTyp := 3;
		PStartSetPlate2.PosTyp := 0;
		
		// Startposition für Ausrichtung von Platten
		PStartAPlate.q1 := 0.175;
		PStartAPlate.q2 := 0.471;
		PStartAPlate.q3 := 0.236;
		PStartAPlate.q4 := 0;
		PStartAPlate.q5 := -180;
		PStartAPlate.q6 := 0;
		PStartAPlate.v := 1;
		PStartAPlate.a := 1;
		PStartAPlate.MoveTyp := 3;
		PStartAPlate.PosTyp := 0;
		
		// Lagerposition von Fixierungsplatte
		PGetFixPlate.q1 := 0.240;
		PGetFixPlate.q2 := 0.5266;
		PGetFixPlate.q3 := 0.243;
		PGetFixPlate.q4 := 3;
		PGetFixPlate.q5 := -180;
		PGetFixPlate.q6 := 0;
		PGetFixPlate.v := 1;
		PGetFixPlate.a := 1;
		PGetFixPlate.MoveTyp := 3;
		PGetFixPlate.PosTyp := 0;
		
		// Startposition für Platzierung von MontagePlatte
		PStartSetFixPlate.q1 := 0.092;
		PStartSetFixPlate.q2 := 0.473;
		PStartSetFixPlate.q3 := 0.246;
		PStartSetFixPlate.q4 := 3;
		PStartSetFixPlate.q5 := -180;
		PStartSetFixPlate.q6 := 0;
		PStartSetFixPlate.v := 1;
		PStartSetFixPlate.a := 1;
		PStartSetFixPlate.MoveTyp := 3;
		PStartSetFixPlate.PosTyp := 0;
		
		// Startposition für Ausrichtung von Fixierplatte in X-Richtung
		PStartAXFixPlate.q1 := 0.211;
		PStartAXFixPlate.q2 := 0.527;
		PStartAXFixPlate.q3 := 0.244;
		PStartAXFixPlate.q4 := 3;
		PStartAXFixPlate.q5 := -180;
		PStartAXFixPlate.q6 := 0;
		PStartAXFixPlate.v := 1;
		PStartAXFixPlate.a := 1;
		PStartAXFixPlate.MoveTyp := 3;
		PStartAXFixPlate.PosTyp := 0;
		
		// Startposition für Ausrichtung von Fixierplatte in Y-Richtung
		PStartAYFixPlate.q1 := 0.2397;
		PStartAYFixPlate.q2 := 0.5037;
		PStartAYFixPlate.q3 := 0.241;
		PStartAYFixPlate.q4 := 3;
		PStartAYFixPlate.q5 := -180;
		PStartAYFixPlate.q6 := 0;
		PStartAYFixPlate.v := 1;
		PStartAYFixPlate.a := 1;
		PStartAYFixPlate.MoveTyp := 3;
		PStartAYFixPlate.PosTyp := 0;
		
		
	// Offsets
		// Offset X (klein - positiv)
		POffsetXs.q1 := 0.02;
		POffsetXs.q2 := 0;
		POffsetXs.q3 := 0;
		POffsetXs.q4 := 0;
		POffsetXs.q5 := 0;
		POffsetXs.q6 := 0;
		POffsetXs.v := 0.02;
		POffsetXs.a := 0.02;
		POffsetXs.MoveTyp := 0;
		POffsetXs.PosTyp := 1;
		
		// Offset X (klein - negativ)
		POffsetnXs.q1 := -0.02;
		POffsetnXs.q2 := 0;
		POffsetnXs.q3 := 0;
		POffsetnXs.q4 := 0;
		POffsetnXs.q5 := 0;
		POffsetnXs.q6 := 0;
		POffsetnXs.v := 0.02;
		POffsetnXs.a := 0.02;
		POffsetnXs.MoveTyp := 0;
		POffsetnXs.PosTyp := 1;
		
		// Offset Y (klein - negativ)
		POffsetnYs.q1 := 0;
		POffsetnYs.q2 := -0.02;
		POffsetnYs.q3 := 0;
		POffsetnYs.q4 := 0;
		POffsetnYs.q5 := 0;
		POffsetnYs.q6 := 0;
		POffsetnYs.v := 0.02;
		POffsetnYs.a := 0.02;
		POffsetnYs.MoveTyp := 0;
		POffsetnYs.PosTyp := 1;
		
		// Z-Richtung (negativ)
		POffsetnZ.q1 := 0;
		POffsetnZ.q2 := 0;
		POffsetnZ.q3 := -0.03;
		POffsetnZ.q4 := 0;
		POffsetnZ.q5 := 0;
		POffsetnZ.q6 := 0;
		POffsetnZ.v := 0.1;
		POffsetnZ.a := 0.1;
		POffsetnZ.MoveTyp := 0;
		POffsetnZ.PosTyp := 1;
		
		// Z-Richtung (positiv)
		POffsetZ.q1 := 0;
		POffsetZ.q2 := 0;
		POffsetZ.q3 := 0.03;
		POffsetZ.q4 := 0;
		POffsetZ.q5 := 0;
		POffsetZ.q6 := 0;
		POffsetZ.v := 0.1;
		POffsetZ.a := 0.1;
		POffsetZ.MoveTyp := 0;
		POffsetZ.PosTyp := 1;
		
	// Ausrichtungs_Offsets
		// Offset X  (positiv)
		POffsetAX.q1 := 0.3;
		POffsetAX.q2 := 0;
		POffsetAX.q3 := 0;
		POffsetAX.q4 := 0;
		POffsetAX.q5 := 0;
		POffsetAX.q6 := 0;
		POffsetAX.v := 0.05;
		POffsetAX.a := 0.05;
		POffsetAX.MoveTyp := 0;
		POffsetAX.PosTyp := 1;
		
		// Offset X für Platte 1 (negativ)
		POffsetAnX.q1 := -0.3;
		POffsetAnX.q2 := 0;
		POffsetAnX.q3 := 0;
		POffsetAnX.q4 := 0;
		POffsetAnX.q5 := 0;
		POffsetAnX.q6 := 0;
		POffsetAnX.v := 0.05;
		POffsetAnX.a := 0.05;
		POffsetAnX.MoveTyp := 0;
		POffsetAnX.PosTyp := 1;
		
		// Offset Y (positiv)
		POffsetAY.q1 := 0;
		POffsetAY.q2 := 0.3;
		POffsetAY.q3 := 0;
		POffsetAY.q4 := 0;
		POffsetAY.q5 := 0;
		POffsetAY.q6 := 0;
		POffsetAY.v := 0.05;
		POffsetAY.a := 0.05;
		POffsetAY.MoveTyp := 0;
		POffsetAY.PosTyp := 1;

		// Offset Y für Platte 1 (negativ)
		POffsetAnY.q1 := 0;
		POffsetAnY.q2 := -0.3;
		POffsetAnY.q3 := 0;
		POffsetAnY.q4 := 0;
		POffsetAnY.q5 := 0;
		POffsetAnY.q6 := 0;
		POffsetAnY.v := 0.01;
		POffsetAnY.a := 0.01;
		POffsetAnY.MoveTyp := 0;
		POffsetAnY.PosTyp := 1;
		
		// Offset Z für Fixierungsplatte (negativ)
		POffsetAnZ.q1 := 0;
		POffsetAnZ.q2 := 0;
		POffsetAnZ.q3 := -0.3;
		POffsetAnZ.q4 := 0;
		POffsetAnZ.q5 := 0;
		POffsetAnZ.q6 := 0;
		POffsetAnZ.v := 0.02;
		POffsetAnZ.a := 0.02;
		POffsetAnZ.MoveTyp := 0;
		POffsetAnZ.PosTyp := 1;

// Greiferpositionen
	// Platte offen
	Plate_Open.Pos := 25;
	Plate_Open.F := 60;
	Plate_Open.Geschw := 20;
	
	// Platte zu
	Plate_Closed.Pos := 15;
	Plate_Closed.F := 60;
	Plate_Closed.Geschw := 20;
	
	// Fixierungsplatte offen
	FixPlate_Open.Pos := 35;
	FixPlate_Open.F := 60;
	FixPlate_Open.Geschw := 20;
	
	// Fixierungsplatte zu
	FixPlate_Closed.Pos := 25;
	FixPlate_Closed.F := 80;
	FixPlate_Closed.Geschw := 20;
	
	// Greifer geschlossen
	GripperClossed.Pos := 0;
	GripperClossed.F := 60;
	GripperClossed.Geschw := 100;

// Kraftvariablen
	// X-Richtung (Bewegungsrichtung: negativ)
	AnstossX.Fx := 0;
	AnstossX.Fy := -5;
	AnstossX.Fz := 0;
	
	// X-Richtung (Bewegungsrichtung: positiv)
	AnstossnX.Fx := 0;
	AnstossnX.Fy := 5;
	AnstossnX.Fz := 0;
	
	// Y-Richtung (Bewegungsrichtung: negativ)
	AnstossY.Fx := -5;
	AnstossY.Fy := 0;
	AnstossY.Fz := 0;
	
	// Y-Richtung (Bewegungsrichtung: positiv)
	AnstossnY.Fx := 5;
	AnstossnY.Fy := 0;
	AnstossnY.Fz := 0;
	
	// Z-Richtung (Bewegungsrichtung: negativ)
	AnstossZ.Fx := 0;
	AnstossZ.Fy := 0;
	AnstossZ.Fz := -20;



// Zuweisung
R_Data_1[0] := PGetPlate1;
R_Data_1[1] := POffsetnZ;
R_Data_1[2] := POffsetZ;

G_Data_1[0] := Plate_Open;
G_Data_1[1] := Plate_Closed;

R_Data_2[0] := PStartSetPlate1;
R_Data_2[1] := POffsetnZ;
R_Data_2[2] := POffsetAnY;
R_Data_2[3] := POffsetAnX;
R_Data_2[4] := POffsetZ;

S_Data_1[0] := AnstossY;
S_Data_1[1] := AnstossX;

R_Data_3[0] := PGetPlate2;
R_Data_3[1] := POffsetnZ;
R_Data_3[2] := POffsetZ;

R_Data_4[0] := PStartSetPlate2;
R_Data_4[1] := POffsetnZ;
R_Data_4[2] := POffsetAnX;
R_Data_4[3] := POffsetZ;

R_Data_5[0] := PStartAPlate;
R_Data_5[1] := POffsetnZ;
R_Data_5[2] := POffsetAnX;
R_Data_5[3] := POffsetXs;
R_Data_5[4] := POffsetZ;

R_Data_6[0] := PStartAXFixPlate;
R_Data_6[1] := POffsetnZ;
R_Data_6[2] := POffsetAX;
R_Data_6[3] := POffsetnXs;
R_Data_6[4] := POffsetZ;

R_Data_7[0] := PStartAYFixPlate;
R_Data_7[1] := POffsetnZ;
R_Data_7[2] := POffsetAY;
R_Data_7[3] := POffsetnYs;
R_Data_7[4] := POffsetZ;

R_Data_8[0] := PGetFixPlate;
R_Data_8[1] := POffsetnZ;
R_Data_8[2] := POffsetZ;

G_Data_2[0] := FixPlate_Open;
G_Data_2[1] := FixPlate_Closed;

R_Data_9[0] := PStartSetFixPlate;
R_Data_9[1] := POffsetAnZ;
R_Data_9[2] := POffsetZ;

END_PROGRAM

// ---- POUs/01_Prozessmodell/03_Arbeitsplan/AP_V2.TcPOU
PROGRAM AP_V2
VAR
	// Bedienparameter
	
	// Prozessparameter
	
	// Skill-Instanziierung
	Skill_R_P2P			:Skill_Position_anfahren;
	Skill_R_Ausrichten	:Skill_Position_anfahren_erweitert;
	Skill_G_P2P			:Skill_Greifer_Pos_Anfahren;
	
	// Sequenz-Instanziierung
	Seq_Get_Teil		:Seq_Teile_Hohlen;
	
	
END_VAR

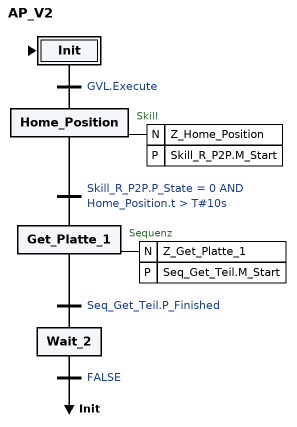
INITIAL_STEP Init:
END_STEP
TRANSITION FROM Init TO Home_Position
    := GVL.Execute;
END_TRANSITION
// Skill
STEP Home_Position:
    Z_Home_Position(N);
    Skill_R_P2P.M_Start(P);
END_STEP
TRANSITION FROM Home_Position TO Get_Platte_1
    := Skill_R_P2P.P_State = 0 AND Home_Position.t > T#10s;
END_TRANSITION
// Sequenz
STEP Get_Platte_1:
    Z_Get_Platte_1(N);
    Seq_Get_Teil.M_Start(P);
END_STEP
TRANSITION FROM Get_Platte_1 TO Wait_2
    := Seq_Get_Teil.P_Finished;
END_TRANSITION
STEP Wait_2:
END_STEP
TRANSITION FROM Wait_2 TO Init
    := FALSE;
END_TRANSITION

ACTION Z_Get_Platte_1:
Seq_Get_Teil(
    eSysCommand := GVL.SystemCommand,
    Param_StartPos := PunkteZuweisung_Temp.PGetPlate1,
    Param_Backenbreite := 20,
    I_Roboter := Anlage.UR5,
    I_Greifer := Anlage.Gripper); // Seq_Teile_Hohlen
END_ACTION

ACTION Z_Home_Position:
Skill_R_P2P(eSysCommand := GVL.SystemCommand,
			eSysState := GVL.SystemState,
			Objekt := Anlage.UR5,
			iErrorID => GVL.ErrorID);

Skill_R_P2P.P_RobotParam := PunkteZuweisung_Temp.PHome;
END_ACTION

ACTION Z_Start_Pos:
// Skillaufruf
Skill_R_P2P(eSysCommand := GVL.SystemCommand,
			eSysState := GVL.SystemState,
			Objekt := Anlage.UR5,
			iErrorID => GVL.ErrorID);

		
// Parameterzuweisung	
Skill_R_P2P.P_RobotParam := PunkteZuweisung_Temp.PGetPlate1;
END_ACTION

END_PROGRAM

// ---- POUs/01_Prozessmodell/01_Skills/02_V2/01_Roboter/Skill_R_P2P.TcPOU
FUNCTION_BLOCK Skill_R_P2P EXTENDS FB_SkillBasis
VAR_INPUT
	// Objekt
	Roboter				:I_Objekt_Roboter;
	
	// Prozessparameter
	Position			:sPositionValues;
	Geschw				:LREAL;
	Beschl				:LREAL;
	PosTyp				:eRobPosType;
	MoveTyp				:eRobMoveType;	
END_VAR
VAR_OUTPUT
END_VAR
VAR
	Prozessparameter	:sRoboterProzessVariablen; 
END_VAR

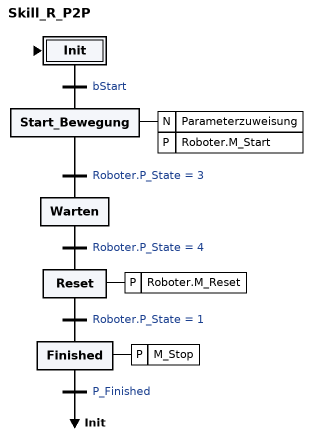
INITIAL_STEP Init:
END_STEP
TRANSITION FROM Init TO Start_Bewegung
    := bStart;
END_TRANSITION
STEP Start_Bewegung:
    Parameterzuweisung(N);
    Roboter.M_Start(P);
END_STEP
TRANSITION FROM Start_Bewegung TO Warten
    := Roboter.P_State = 3;
END_TRANSITION
STEP Warten:
END_STEP
TRANSITION FROM Warten TO Reset
    := Roboter.P_State = 4;
END_TRANSITION
STEP Reset:
    Roboter.M_Reset(P);
END_STEP
TRANSITION FROM Reset TO Finished
    := Roboter.P_State = 1;
END_TRANSITION
STEP Finished:
    M_Stop(P);
END_STEP
TRANSITION FROM Finished TO Init
    := P_Finished;
END_TRANSITION

ACTION Parameterzuweisung:
// Variablenzuweisung
Prozessparameter.q1 := Position.q1;
Prozessparameter.q2 := Position.q2;
Prozessparameter.q3 := Position.q3;
Prozessparameter.q4 := Position.q4;
Prozessparameter.q5 := Position.q5;
Prozessparameter.q6 := Position.q6;
Prozessparameter.v := Geschw;
Prozessparameter.a := Beschl;
Prozessparameter.MoveTyp := MoveTyp;
Prozessparameter.PosTyp := PosTyp;

//Zuweisung an Objekt
Roboter.P_Prozessparameter := Prozessparameter;
END_ACTION

END_FUNCTION_BLOCK

// ---- POUs/01_Prozessmodell/01_Skills/02_V2/01_Roboter/FB_SkillBasis.TcPOU
FUNCTION_BLOCK FB_SkillBasis
VAR_INPUT
	
END_VAR
VAR_OUTPUT
END_VAR
VAR
	// Interne Variablen
	bStart					:BOOL;
	bStop					:BOOL;
	
	// SFC-Flags
	SFCReset				:BOOL;
END_VAR

METHOD M_Reset : BOOL
VAR_INPUT
END_VAR
bStart := FALSE;
bStop := FALSE; 
SFCReset := TRUE;
END_METHOD

METHOD M_Start : BOOL
VAR_INPUT
END_VAR
SFCReset := FALSE;
bStop := FALSE;
bStart := TRUE;
END_METHOD

METHOD M_Stop : BOOL
VAR_INPUT
END_VAR
bStart := FALSE; 
bStop := TRUE;
END_METHOD

PROPERTY P_Finished : BOOL
GET
P_Finished := bStop;
END_GET
END_PROPERTY

END_FUNCTION_BLOCK

// ---- POUs/01_Prozessmodell/01_Skills/01_V1/01_Roboter/Skill_Position_anfahren.TcPOU
FUNCTION_BLOCK Skill_Position_anfahren EXTENDS FB_Basis_Skill IMPLEMENTS I_Skill_Roboter
VAR_INPUT
	// Zu verwendetes Objekt
	Objekt						:I_Objekt_Roboter;	
END_VAR
VAR_OUTPUT
END_VAR
VAR
	// Prozessparameter
	eRoboterPos		 			:sRoboterProzessVariablen;
	
	// Test
	bPulseNr					:INT;
END_VAR

// Parameterzuweisung
Objekt.P_Prozessparameter := eRoboterPos;

// Fehlerüberwachung
IF bFehler THEN
	iState := 3;
END_IF

//_______________________________________________________________
// Reaktion auf Input-Variablen:
	// Stoppen
	IF eSysCommand = 3 THEN
		bStoppen := M_Stop();
	ELSE 
		bStoppen := FALSE;
	END_IF

	// Resetten 
	IF eSysCommand = 4 THEN
		bResetten := M_Reset();
	ELSE
		bResetten := FALSE;
	END_IF
//_______________________________________________________________
// Zustandsmanagement
CASE iState OF 
0: 	// BEREIT	
		// DO
		IF Objekt.P_State = 3 AND bSkillActiv THEN		// Objekt wurde eingeschalten
			bStarten := TRUE;
		END_IF
		
		// TRANSITION
		IF bStarten	 THEN		
			bStarten := FALSE;
			iState := 1;	
		END_IF
// _________________________________________________________________________________________________________________________
1: 	// LAUFEND
		// DO			
			// Stoppen durch Sysezm
			IF bStoppen THEN																								// Transition wenn System das Orbjekt stoppt
				bGestoppt := TRUE;
			END_IF
			
			// Objekt hat sich selber gestoppt
			IF Objekt.P_State = 4 THEN																							// Objekt hat Prozess abgeschlossen
				bObjektFertig := TRUE;																							// Objekt ist fertig und wieder bereit
			END_IF
			
		// TRANSITION 
		IF bGestoppt THEN																								// Transition zu BEREIT
			bGestoppt := FALSE;																					
			iState := 0;
		END_IF
		
		IF bObjektFertig THEN																							// Transition zu ABGESCHLOSSEN
			bObjektFertig := FALSE;																							// Skill wird nicht mehr ausgeführt
			iState := 2;																									// Objekt ist fertig und wieder bereit
		END_IF
		
		IF bLimitErreicht AND Objekt.P_State = 5 THEN																							// Transition zu LIMIT
			iState := 4;
		END_IF
		
		IF bWertErreicht AND Objekt.P_State = 5 THEN																							// Transition zu ERREICHT
			iState := 5;
		END_IF			
// _________________________________________________________________________________________________________________________			
2: 	// ABGESCHLOSSEN
		// DO
		M_Reset();
		
		IF Objekt.P_State = 1 THEN																							// Objekt wurde geresettet
			bSkillFertig := TRUE;									
		END_IF
			
		//  TRANSITION
		IF bSkillFertig THEN
			bSkillFertig := FALSE;																																											// Resetten von Objekt
			iState := 0;
		END_IF
// _________________________________________________________________________________________________________________________
3: 	// FEHLER
		// DO 	
		IF ParameterError THEN
			// Setzen von ErrorID
		END_IF
		
		IF PositionError THEN
			// Setzen von ErrorID
		END_IF
		
		// TRANSITION
		IF bResetten THEN
			bFehler := FALSE;
			iState := 0;
		END_IF
		
END_CASE

IF GVL.skillInfo[GVL.InfoCountSkill].iState <> iState THEN
	GVL.InfoCountSkill := GVL.InfoCountSkill + 1;
	GVL.skillInfo[GVL.InfoCountSkill].iState := iState;
	GVL.skillInfo[GVL.InfoCountSkill].iStateObj := Objekt.P_State;
	GVL.skillInfo[GVL.InfoCountSkill].Data := eRoboterPos;
	GVL.skillInfo[GVL.InfoCountSkill].DataObj := Objekt.Test_Param;
END_IF 

GVL.TestCount := GVL.TestCount + 1;

METHOD M_Reset : BOOL
Objekt.M_Reset();
bSkillActiv := FALSE;
END_METHOD

METHOD M_Start : BOOL
GVL.CountSkillStart := GVL.CountSkillStart + 1;
// Ausführen von Funktion
GVL.MethodeState := 0;
IF NOT bSkillActiv THEN
	GVL.MethodeState := 1;
	// Ist das  System im korrekten Status
	IF eSysState = 1 OR eSysState = 2 THEN
		GVL.MethodeState := 2;
		// Ist der Skill im korrekten Status 
		IF iState = 0 THEN
			GVL.MethodeState := 3;
			// Prüfen auf Fehler
			IF ParameterError OR PositionError THEN
				bFehler := TRUE;
			ELSE
				GVL.MethodeState := 4;
				Objekt.M_Start();
				bSkillActiv := TRUE;
				GVL.SkillArray[GVL.CountSkill] := eRoboterPos;
				GVL.CountSkill := GVL.CountSkill + 1;
			END_IF
		END_IF
	END_IF
END_IF
END_METHOD

METHOD M_Stop : BOOL

Objekt.M_Stop();
bSkillActiv := FALSE;
END_METHOD

PROPERTY P_RobotParam : sRoboterProzessVariablen
SET
eRoboterPos := P_RobotParam;
END_SET
END_PROPERTY

PROPERTY P_State : eSkillState
GET
P_State := iState;
END_GET
END_PROPERTY

TRANSITION ParameterError:
IF eRoboterPos.a = 0 OR eRoboterPos.v = 0 THEN
	ParameterError := TRUE;
END_IF
END_TRANSITION

TRANSITION PositionError:
IF eRoboterPos.q1 = 0 AND eRoboterPos.q2 = 0 AND eRoboterPos.q3 = 0 AND eRoboterPos.q4 = 0 AND eRoboterPos.q5 = 0 AND eRoboterPos.q6 = 0 THEN
	PositionError := TRUE;
END_IF
END_TRANSITION

END_FUNCTION_BLOCK

// ---- POUs/01_Prozessmodell/01_Skills/01_V1/00_Basis/FB_Basis_Skill.TcPOU
FUNCTION_BLOCK FB_Basis_Skill
VAR_INPUT
	// Betriebsvariablen 
	eSysCommand					:eSystemCommand; 						// Systembefehl an Skill
	eSysState					:eSystemState;							// Momentaner Zustand des Systems
END_VAR
VAR_OUTPUT
	iErrorID					:INT;									// Fehlercode für System
END_VAR
VAR
	// Managementvariablen
	iState						:eSkillState;							// Information über Zustand von Skill
	
	bGestartet					:BOOL;									// Skill wurde gestartet
	bGestoppt					:BOOL;									// Skill wurde gestoppt
	bSkillActiv					:BOOL;									// Skill ist im Moment aktiv
	
	// Zustandsvariablen (Transitions)
	bStarten					:BOOL;									
	bStoppen					:BOOL;
	bObjektFertig				:BOOL;
	bWertErreicht				:BOOL;				
	bLimitErreicht				:BOOL;				
	bSkillFertig				:BOOL;
	bFehler						:BOOL;
	bResetten					:BOOL;
	bErreicht					:BOOL;				
	bLimit						:BOOL;
END_VAR

END_FUNCTION_BLOCK

// ---- POUs/01_Prozessmodell/02_Sequenzen/02_Version_2/Seq_Teile_Hohlen.TcPOU

FUNCTION_BLOCK Seq_Teile_Hohlen EXTENDS FB_Basis
VAR_INPUT
	// Prozessparameter		
	Param_StartPos				:sRoboterProzessVariablen;
	Param_Backenbreite			:USINT;
	
	// Objekt-Schnittstellen
	I_Roboter					:I_Objekt_Roboter;
	I_Greifer					:I_Objekt_SmartGreifer;	
END_VAR
VAR_OUTPUT
END_VAR
VAR
	// Skill-Instanziierung
	Skill_R_P2P				:Skill_Position_anfahren;
	Skill_G_P2P				:Skill_Greifer_Pos_Anfahren;
	
	// Interne Prozessvariablen
	LRobotVar				:sRoboterProzessVariablen;
	LGreiferVar				:sSmartGreiferProzessVariablen;
	LOffsetVar				:LREAL;
END_VAR


// Ablauf
ACT_Ablauf();

// Zustandshandling
CASE iState OF
	0:	// BEREIT
		IF bStart THEN
			iState := 1;
		END_IF
	1:	// LAUFEND
		IF eSysCommand = 4 THEN
			bReset := TRUE;
			SFCReset := TRUE;
		END_IF
		
		IF bBeendet OR bReset THEN
			bReset := FALSE;
			SFCReset := FALSE;
			iState := 0;
		END_IF
	2: // ABGESCHLOSSEN
		IF SFCCurrentStep = 'Init' THEN
			iState := 0;
		END_IF
END_CASE

ACTION ACT_Ablauf:
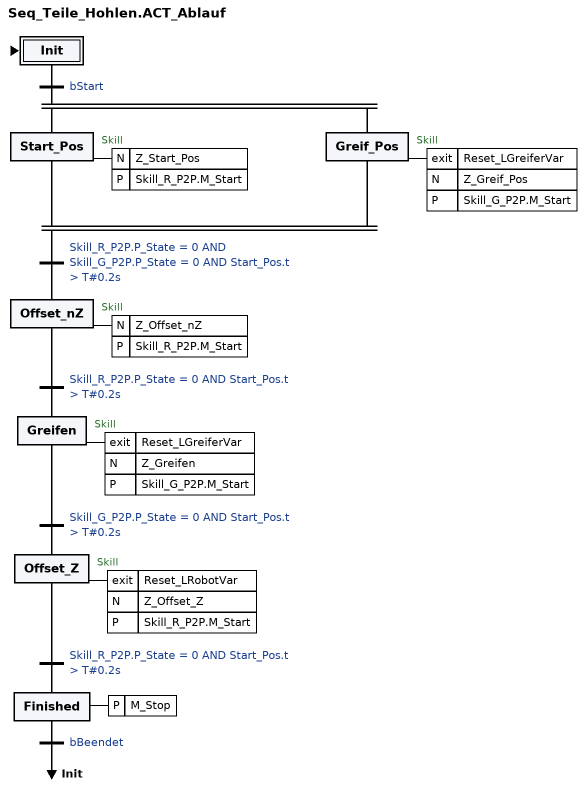
INITIAL_STEP Init:
END_STEP
TRANSITION FROM Init TO (Start_Pos, Greif_Pos)
    := bStart;
END_TRANSITION
// Skill
STEP Start_Pos:
    Z_Start_Pos(N);
    Skill_R_P2P.M_Start(P);
END_STEP
// Skill
STEP Greif_Pos:
    Reset_LGreiferVar(P0);  // exit action
    Z_Greif_Pos(N);
    Skill_G_P2P.M_Start(P);
END_STEP
TRANSITION FROM (Start_Pos, Greif_Pos) TO Offset_nZ
    := Skill_R_P2P.P_State = 0 AND Skill_G_P2P.P_State = 0 AND Start_Pos.t > T#0.2s;
END_TRANSITION
// Skill
STEP Offset_nZ:
    Z_Offset_nZ(N);
    Skill_R_P2P.M_Start(P);
END_STEP
TRANSITION FROM Offset_nZ TO Greifen
    := Skill_R_P2P.P_State = 0 AND Start_Pos.t > T#0.2s;
END_TRANSITION
// Skill
STEP Greifen:
    Reset_LGreiferVar(P0);  // exit action
    Z_Greifen(N);
    Skill_G_P2P.M_Start(P);
END_STEP
TRANSITION FROM Greifen TO Offset_Z
    := Skill_G_P2P.P_State = 0 AND Start_Pos.t > T#0.2s;
END_TRANSITION
// Skill
STEP Offset_Z:
    Reset_LRobotVar(P0);  // exit action
    Z_Offset_Z(N);
    Skill_R_P2P.M_Start(P);
END_STEP
TRANSITION FROM Offset_Z TO Finished
    := Skill_R_P2P.P_State = 0 AND Start_Pos.t > T#0.2s;
END_TRANSITION
STEP Finished:
    M_Stop(P);
END_STEP
TRANSITION FROM Finished TO Init
    := bBeendet;
END_TRANSITION
END_ACTION

ACTION Reset_LGreiferVar:
LGreiferVar.F := 0;
LGreiferVar.Geschw := 0;
LGreiferVar.Pos := 0;
END_ACTION

ACTION Reset_LRobotVar:
LRobotVar.q1 := 0;
LRobotVar.q2 := 0;
LRobotVar.q3 := 0;
LRobotVar.q4 := 0;
LRobotVar.q5 := 0;
LRobotVar.q6 := 0;
LRobotVar.v := 0;
LRobotVar.a := 0;
LRobotVar.MoveTyp := 0;
LRobotVar.PosTyp := 0;
END_ACTION

ACTION Z_Greif_Pos:
// Skillaufruf
Skill_G_P2P(eSysCommand := GVL.SystemCommand,
			eSysState := GVL.SystemState,
			Objekt := I_Greifer,
			iErrorID => GVL.ErrorID);
			
// Parameterbestimmung
LGreiferVar.F := 100;
LGreiferVar.Geschw := 100;
LGreiferVar.Pos := Param_Backenbreite;		

// Parameterzuweisung
Skill_G_P2P.P_SGripperParam := LGreiferVar;
END_ACTION

ACTION Z_Greifen:
// Skillaufruf
Skill_G_P2P(eSysCommand := GVL.SystemCommand,
			eSysState := GVL.SystemState,
			Objekt := I_Greifer,
			iErrorID => GVL.ErrorID);
			
// Parameterbestimmung
LGreiferVar.F := 50;
LGreiferVar.Geschw := 50;
LGreiferVar.Pos := 10;		

// Parameterzuweisung
Skill_G_P2P.P_SGripperParam := LGreiferVar;
END_ACTION

ACTION Z_Home_Position_:
// Skillaufruf
Skill_R_P2P(eSysCommand := GVL.SystemCommand,
			eSysState := GVL.SystemState,
			Objekt := I_Roboter,
			iErrorID => GVL.ErrorID);


// Parameterbestimmung			
LRobotVar := PunkteZuweisung_Temp.PHome;
		
// Parameterzuweisung	
Skill_R_P2P.P_RobotParam := LRobotVar;
END_ACTION

ACTION Z_Offset_nZ:
// Skillaufruf
Skill_R_P2P(eSysCommand := GVL.SystemCommand,
			eSysState := GVL.SystemState,
			Objekt := I_Roboter,
			iErrorID => GVL.ErrorID);

// Parameterbestimmung			
LRobotVar.q1 := 0;
LRobotVar.q2 := 0;
LRobotVar.q3 := -0.03;
LRobotVar.q4 := 0;
LRobotVar.q5 := 0;
LRobotVar.q6 := 0;
LRobotVar.v := 0.1;
LRobotVar.a := 0.1;
LRobotVar.MoveTyp := 0;
LRobotVar.PosTyp := 1;

// Parameterzuweisung	
Skill_R_P2P.P_RobotParam := LRobotVar;
END_ACTION

ACTION Z_Offset_Z:
// Skillaufruf
Skill_R_P2P(eSysCommand := GVL.SystemCommand,
			eSysState := GVL.SystemState,
			Objekt := I_Roboter,
			iErrorID => GVL.ErrorID);

// Parameterbestimmung			
LRobotVar.q1 := 0;
LRobotVar.q2 := 0;
LRobotVar.q3 := 0.03;
LRobotVar.q4 := 0;
LRobotVar.q5 := 0;
LRobotVar.q6 := 0;
LRobotVar.v := 0.1;
LRobotVar.a := 0.1;
LRobotVar.MoveTyp := 0;
LRobotVar.PosTyp := 1;
		
// Parameterzuweisung	
Skill_R_P2P.P_RobotParam := LRobotVar;
END_ACTION

ACTION Z_Start_Pos:

// Skillaufruf
Skill_R_P2P(eSysCommand := GVL.SystemCommand,
			eSysState := GVL.SystemState,
			Objekt := I_Roboter,
			iErrorID => GVL.ErrorID);

// Parameterbestimmung			
LRobotVar := Param_StartPos;
		
// Parameterzuweisung	
Skill_R_P2P.P_RobotParam := LRobotVar;
END_ACTION

END_FUNCTION_BLOCK

// ---- POUs/01_Prozessmodell/02_Sequenzen/00_Basis/FB_Basis.TcPOU
FUNCTION_BLOCK FB_Basis
VAR_INPUT
	// Betriebsvariablen
	eSysCommand				:eSystemCommand;
END_VAR
VAR_OUTPUT
END_VAR
VAR
	// Managementvariablen
	iState					:INT;
	
	// Transitionsvariablen
	bStart					:BOOL;
	bBeendet 				:BOOL;
	bReset					:BOOL;
	
	// SFC-Flags
	SFCReset				:BOOL;
	SFCCurrentStep			:BOOL;
END_VAR

METHOD M_Reset : BOOL
VAR_INPUT
END_VAR
bReset := TRUE;
END_METHOD

METHOD M_Start : BOOL
VAR_INPUT
END_VAR
// Prüfen ob sich Sequenz im korrekten Zustand befindet
IF iState = 0 THEN
	bBeendet := FALSE;
	bStart := TRUE;
END_IF
END_METHOD

METHOD M_Stop : BOOL
VAR_INPUT
END_VAR
bStart := FALSE;
bBeendet := TRUE;
END_METHOD

PROPERTY P_Finished : BOOL
GET
P_Finished := bBeendet;
END_GET
END_PROPERTY

PROPERTY P_State : INT;
GET
P_State := iState;
END_GET
END_PROPERTY

END_FUNCTION_BLOCK

// ---- POUs/00_Funktionsbausteine/FB_PulseTrigger.TcPOU
FUNCTION_BLOCK FB_PulseTrigger
VAR_INPUT
	Pulse			:BOOL;
END_VAR
VAR_OUTPUT
	Q				:BOOL;
END_VAR
VAR
	Trigger			:R_Trig; 
	Counter			:INT;
END_VAR

IF Pulse THEN
	Trigger(CLK := TRUE);
ELSE
	Trigger(CLK := FALSE);
END_IF

IF Trigger.Q THEN
	Counter := Counter + 1;
END_IF

IF Counter = 1 THEN
	Q := TRUE;
END_IF
IF Counter = 2 THEN
	Q := FALSE;
	Counter := 0;
END_IF

END_FUNCTION_BLOCK

// ---- POUs/01_Prozessmodell/01_Skills/01_V1/00_Basis/FB_SkillReferenz.TcPOU
FUNCTION_BLOCK FB_SkillReferenz EXTENDS FB_Basis_Skill IMPLEMENTS I_Skill 
VAR_INPUT
	// Zu verwendetes Objekt
	Objekt						:I_Objekt_Roboter;	
	
	// Prozessrelevante Inputs
	sMessdaten					:Kraftvariablen; 
END_VAR
VAR_OUTPUT
	iErrorID					:INT;									// Fehlercode für System
END_VAR
VAR
	// Prozessvariablen
	eProzessvariable 	:sRoboterProzessVariablen;
END_VAR

// Fehlerüberwachung
IF bFehler THEN
	iState := 3;
END_IF

//_______________________________________________________________
// Interner Steuerungsmethodenaufruf:
	// Stoppen
	IF eSysCommand = 3 THEN
		bStoppen := M_Stop();
	ELSE 
		bStoppen := FALSE;
	END_IF

	// Resetten 
	IF eSysCommand = 4 THEN
		bResetten := M_Reset();
	ELSE
		bResetten := FALSE;
	END_IF
	
	// Limit
	IF bLimit THEN
		bLimitErreicht := M_Stop();
	ELSE
		bLimitErreicht := FALSE;
	END_IF
	
	// Erreicht
	IF bErreicht THEN
		bWertErreicht := M_Stop();
	ELSE
		bWertErreicht := FALSE;
	END_IF
//_______________________________________________________________
// Zustandsmanagement
CASE iState OF 
0: 	// BEREIT	
		// DO
		IF Objekt.P_State = 3 THEN		// Objekt wurde eingeschalten
			bStarten := TRUE;
		END_IF
		
		// TRANSITION
		IF bStarten	 THEN		
			bStarten := FALSE;
			iState := 1;	
		END_IF
		
		
// _________________________________________________________________________________________________________________________
1: 	// LAUFEND
		// DO			
			// Stoppen durch Sysezm
			IF bStoppen THEN																								// Transition wenn System das Orbjekt stoppt
				bGestoppt := TRUE;
			END_IF
			
			// Objekt hat sich selber gestoppt
			IF Objekt.P_State = 4 THEN																							// Objekt hat Prozess abgeschlossen
				bObjektFertig := TRUE;																							// Objekt ist fertig und wieder bereit
			END_IF
			
		// TRANSITION 
		IF bGestoppt THEN																								// Transition zu BEREIT
			bGestoppt := FALSE;																						
			iState := 0;
		END_IF
		
		IF bObjektFertig THEN																							// Transition zu ABGESCHLOSSEN
			bObjektFertig := FALSE;																							// Skill wird nicht mehr ausgeführt
			iState := 2;																									// Objekt ist fertig und wieder bereit
		END_IF
		
		IF bLimitErreicht AND Objekt.P_State = 5 THEN																							// Transition zu LIMIT
			iState := 4;
		END_IF
		
		IF bWertErreicht AND Objekt.P_State = 5 THEN																							// Transition zu ERREICHT	
			iState := 5;
		END_IF
			
// _________________________________________________________________________________________________________________________			
2: 	// ABGESCHLOSSEN
		// DO
		IF Objekt.P_State = 1 THEN																							// Objekt wurde geresettet
			bSkillFertig := TRUE;									
		END_IF
			
		//  TRANSITION
		IF bSkillFertig THEN
			bSkillFertig := FALSE;																																											// Resetten von Objekt
			iState := 0;
		END_IF
		
// _________________________________________________________________________________________________________________________
3: 	// FEHLER
		// DO 	
		
		// TRANSITION
		IF bResetten THEN
			iState := 0;
		END_IF
		
// _________________________________________________________________________________________________________________________			
4: 	// LIMIT
		// DO		
		M_Reset();
		
		IF Objekt.P_State = 1 THEN																								// Objekt wurde geresettet
			bResetten := TRUE;								
		END_IF
	
		// TRANSITION
		IF bResetten THEN
			bResetten := FALSE;
			iState := 0;
		END_IF
			
// _________________________________________________________________________________________________________________________
5: 	// ERREICHT		
		// DO 
		M_Reset();
		
		IF Objekt.P_State = 1 THEN																							// Objekt wurde geresettet
			bSkillFertig := TRUE;									
		END_IF
		
		// TRANSITION
		IF bSkillFertig THEN
			bSkillFertig := FALSE;
			iState := 0;
		END_IF
		
END_CASE

METHOD M_Reset : BOOL
Objekt.M_Reset();
END_METHOD

METHOD M_Start : BOOL
// Prüfen von Bedingungen
	// Ist das  System im korrekten Status
	IF eSysState = 1 THEN
		// Ist der Skill im korrekten Status 
		IF iState = 0 THEN
			// Prüfen auf Fehler (Muss ergänzt werden)
				Objekt.P_Prozessparameter := eProzessvariable;
				Objekt.M_Start();
		END_IF
	END_IF
END_METHOD

METHOD M_Stop : BOOL
Objekt.M_Stop();
END_METHOD

PROPERTY P_State : eSkillState
GET
P_State := iState;
END_GET
END_PROPERTY

END_FUNCTION_BLOCK

// ---- POUs/01_Prozessmodell/02_Sequenzen/01_Version_1/Seq_Ausrichten.TcPOU
FUNCTION_BLOCK Seq_Ausrichten EXTENDS FB_Basis IMPLEMENTS I_Sequenz
VAR_INPUT
	// Skillzuweisung
	R_Move					:I_Skill_RoboterErweitert;
	
	// Prozessparameter		
	RobParam				:ARRAY[0..1] OF sRoboterProzessVariablen;
	ErreichtParam			:sKraftVariablen;
END_VAR
VAR_OUTPUT
END_VAR
VAR
	ErreichtParamReset		:sKraftVariablen;
	Counter			:INT;
END_VAR

// Ablauf
ACT_Ablauf();

// Zustandshandling
CASE iState OF
	0:	// BEREIT
		IF bStart THEN
			iState := 1;
		END_IF
	1:	// LAUFEND
		IF eSysCommand = 4 THEN
			bReset := TRUE;
			SFCReset := TRUE;
		END_IF
		
		IF bBeendet OR bReset THEN
			bReset := FALSE;
			SFCReset := FALSE;
			iState := 0;
		END_IF
	2: // ABGESCHLOSSEN
		IF SFCCurrentStep = 'Init' THEN
			iState := 0;
		END_IF
END_CASE

ACTION ACT_Ablauf:
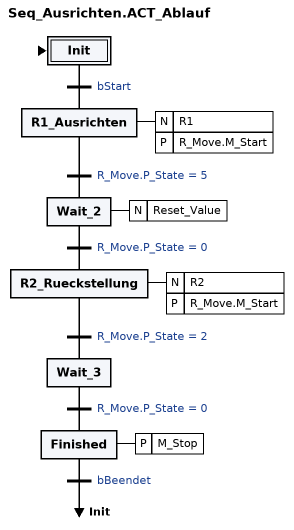
INITIAL_STEP Init:
END_STEP
TRANSITION FROM Init TO R1_Ausrichten
    := bStart;
END_TRANSITION
STEP R1_Ausrichten:
    R1(N);
    R_Move.M_Start(P);
END_STEP
TRANSITION FROM R1_Ausrichten TO Wait_2
    := R_Move.P_State = 5;
END_TRANSITION
STEP Wait_2:
    Reset_Value(N);
END_STEP
TRANSITION FROM Wait_2 TO R2_Rueckstellung
    := R_Move.P_State = 0;
END_TRANSITION
STEP R2_Rueckstellung:
    R2(N);
    R_Move.M_Start(P);
END_STEP
TRANSITION FROM R2_Rueckstellung TO Wait_3
    := R_Move.P_State = 2;
END_TRANSITION
STEP Wait_3:
END_STEP
TRANSITION FROM Wait_3 TO Finished
    := R_Move.P_State = 0;
END_TRANSITION
STEP Finished:
    M_Stop(P);
END_STEP
TRANSITION FROM Finished TO Init
    := bBeendet;
END_TRANSITION
END_ACTION

ACTION R1:
R_Move.P_RobotParam := RobParam[0];
R_Move.P_Erreicht := ErreichtParam;
END_ACTION

ACTION R2:
R_Move.P_RobotParam := RobParam[1];
END_ACTION

ACTION Reset_Value:
ErreichtParamReset.Fx := 0;
ErreichtParamReset.Fy := 0;
ErreichtParamReset.Fz := 0;

R_Move.P_Erreicht := ErreichtParamReset;
END_ACTION

END_FUNCTION_BLOCK

// ---- POUs/01_Prozessmodell/02_Sequenzen/01_Version_1/Seq_Ausrichten_MPlate.TcPOU
FUNCTION_BLOCK Seq_Ausrichten_MPlate EXTENDS FB_Basis IMPLEMENTS I_Sequenz
VAR_INPUT
	// Skillzuweisung
	R_Move					:I_Skill_RoboterErweitert;
	G_Move					:I_Skill_SmartGreifer;
	
	// Prozessparameter		
	RobParam				:ARRAY[0..4] OF sRoboterProzessVariablen;
	GripParam				:sSmartGreiferProzessVariablen;
	ErreichtParam			:sKraftVariablen;
END_VAR
VAR_OUTPUT
END_VAR
VAR
	// Interne Sequenzen
	Seq_Ausrichten			:Seq_Ausrichten;	

	// Interne Paramater 
	Ausrichten_Pos			:ARRAY[0..1] OF sRoboterProzessVariablen;
	ErreichtParamReset		:sKraftVariablen;
END_VAR

// Ablauf
ACT_Ablauf();

// Zustandshandling
CASE iState OF
	0:	// BEREIT
		IF bStart THEN
			iState := 1;
		END_IF
	1:	// LAUFEND
		IF eSysCommand = 4 THEN
			bReset := TRUE;
			SFCReset := TRUE;
		END_IF
		
		IF bBeendet OR bReset THEN
			bReset := FALSE;
			SFCReset := FALSE;
			iState := 0;
		END_IF
	2: // ABGESCHLOSSEN
		IF SFCCurrentStep = 'Init' THEN
			iState := 0;
		END_IF
END_CASE

ACTION ACT_Ablauf:
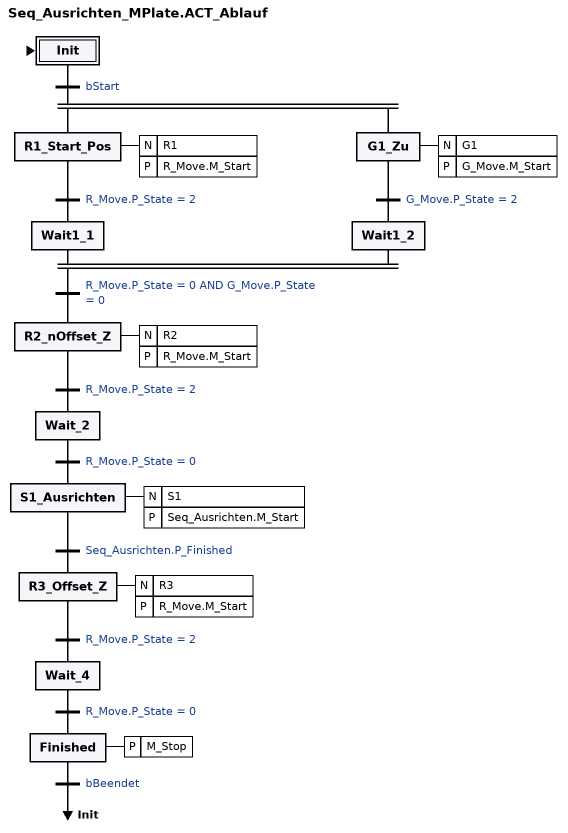
INITIAL_STEP Init:
END_STEP
TRANSITION FROM Init TO (R1_Start_Pos, G1_Zu)
    := bStart;
END_TRANSITION
STEP R1_Start_Pos:
    R1(N);
    R_Move.M_Start(P);
END_STEP
TRANSITION FROM R1_Start_Pos TO Wait1_1
    := R_Move.P_State = 2;
END_TRANSITION
STEP Wait1_1:
END_STEP
STEP G1_Zu:
    G1(N);
    G_Move.M_Start(P);
END_STEP
TRANSITION FROM G1_Zu TO Wait1_2
    := G_Move.P_State = 2;
END_TRANSITION
STEP Wait1_2:
END_STEP
TRANSITION FROM (Wait1_1, Wait1_2) TO R2_nOffset_Z
    := R_Move.P_State = 0 AND G_Move.P_State = 0;
END_TRANSITION
STEP R2_nOffset_Z:
    R2(N);
    R_Move.M_Start(P);
END_STEP
TRANSITION FROM R2_nOffset_Z TO Wait_2
    := R_Move.P_State = 2;
END_TRANSITION
STEP Wait_2:
END_STEP
TRANSITION FROM Wait_2 TO S1_Ausrichten
    := R_Move.P_State = 0;
END_TRANSITION
STEP S1_Ausrichten:
    S1(N);
    Seq_Ausrichten.M_Start(P);
END_STEP
TRANSITION FROM S1_Ausrichten TO R3_Offset_Z
    := Seq_Ausrichten.P_Finished;
END_TRANSITION
STEP R3_Offset_Z:
    R3(N);
    R_Move.M_Start(P);
END_STEP
TRANSITION FROM R3_Offset_Z TO Wait_4
    := R_Move.P_State = 2;
END_TRANSITION
STEP Wait_4:
END_STEP
TRANSITION FROM Wait_4 TO Finished
    := R_Move.P_State = 0;
END_TRANSITION
STEP Finished:
    M_Stop(P);
END_STEP
TRANSITION FROM Finished TO Init
    := bBeendet;
END_TRANSITION
END_ACTION

ACTION G1:
G_Move.P_SGripperParam := GripParam;
END_ACTION

ACTION R1:
R_Move.P_RobotParam := RobParam[0];
END_ACTION

ACTION R2:
R_Move.P_RobotParam := RobParam[1];
END_ACTION

ACTION R3:
R_Move.P_RobotParam := RobParam[4];
END_ACTION

ACTION S1:
Ausrichten_Pos[0] := RobParam[2];
Ausrichten_Pos[1] := RobParam[3];

Seq_Ausrichten(	eSysCommand := GVL.SystemCommand,
				R_Move := SkillSet.Move_2P2_Advanced,
				RobParam := Ausrichten_Pos,
				ErreichtParam := ErreichtParam);
END_ACTION

END_FUNCTION_BLOCK

// ---- POUs/01_Prozessmodell/SkillSet.TcPOU
PROGRAM SkillSet
VAR_INPUT
	Move_2P2			:Skill_Position_anfahren;
	Move_2P2_Advanced	:Skill_Position_anfahren_erweitert;
	
	Grip_2P2			:Skill_Greifer_Pos_Anfahren;
END_VAR

Move_2P2(Objekt := Anlage.UR5, eSysCommand := GVL.SystemCommand, eSysState := GVL.SystemState); // Skill_Position_anfahren
GVL.ErrorID := Move_2P2.iErrorID;
Grip_2P2(Objekt := Anlage.Gripper, eSysCommand := GVL.SystemCommand, eSysState := GVL.SystemState); // Skill_Greifer_Pos_Anfahren
GVL.ErrorID := Grip_2P2.iErrorID;
Move_2P2_Advanced(
    Objekt := Anlage.UR5,
    eSysCommand := GVL.SystemCommand,
    eSysState := GVL.SystemState,
    sMessdaten := Anlage.HEX_E_V2.P_Messdaten); // Skill_Position_anfahren_erweitert
GVL.ErrorID := Move_2P2_Advanced.iErrorID;

END_PROGRAM

// ---- POUs/01_Prozessmodell/02_Sequenzen/01_Version_1/Seq_Ausrichten_Plates.TcPOU
FUNCTION_BLOCK Seq_Ausrichten_Plates EXTENDS FB_Basis IMPLEMENTS I_Sequenz
VAR_INPUT
	// Skillzuweisung
	R_Move			:I_Skill_RoboterErweitert;
	
	// Prozessparameter		
	RobParam				:ARRAY[0..4] OF sRoboterProzessVariablen;
	ErreichtParam			:sKraftVariablen;
END_VAR
VAR_OUTPUT
END_VAR
VAR
	ErreichtParamReset		:sKraftVariablen;
END_VAR

// Ablauf
ACT_Ablauf();

// Zustandshandling
CASE iState OF
	0:	// BEREIT
		IF bStart THEN
			iState := 1;
		END_IF
	1:	// LAUFEND
		IF eSysCommand = 4 THEN
			bReset := TRUE;
			SFCReset := TRUE;
		END_IF
		
